C07304=1154.950,50.044,-50.253,-179.701,6.264,149.045
C07305=1154.955,49.796,-50.237,-179.703,6.263,149.046
C07306=1154.960,49.546,-50.222,-179.706,6.262,149.047
C07307=1154.965,49.296,-50.206,-179.708,6.261,149.047
C07308=1154.970,49.047,-50.190,-179.711,6.260,149.048
C07309=1154.975,48.798,-50.175,-179.714,6.259,149.048
C07310=1154.979,48.548,-50.159,-179.716,6.258,149.049
C07311=1154.985,48.298,-50.144,-179.719,6.257,149.049
C07312=1154.990,48.049,-50.128,-179.721,6.256,149.050
C07313=1154.996,47.800,-50.112,-179.724,6.255,149.050
C07314=1155.000,47.550,-50.097,-179.726,6.254,149.051
C07315=1155.005,47.300,-50.081,-179.730,6.252,149.051
C07316=1155.010,47.051,-50.066,-179.732,6.252,149.052
C07317=1155.015,46.802,-50.051,-179.734,6.251,149.052
C07318=1155.020,46.552,-50.035,-179.737,6.249,149.053
C07319=1155.025,46.302,-50.019,-179.739,6.249,149.053
C07320=1155.030,46.053,-50.004,-179.743,6.247,149.054
C07321=1155.035,45.804,-49.989,-179.745,6.246,149.055
C07322=1155.040,45.554,-49.973,-179.747,6.246,149.055
C07323=1155.045,45.305,-49.958,-179.750,6.244,149.056
C07324=1155.050,45.055,-49.942,-179.753,6.244,149.056
C07325=1155.055,44.806,-49.927,-179.756,6.242,149.057
C07326=1155.060,44.557,-49.912,-179.758,6.241,149.057
C07327=1155.065,44.307,-49.896,-179.760,6.241,149.058
C07328=1155.070,44.057,-49.880,-179.763,6.239,149.058
C07329=1155.075,43.808,-49.865,-179.766,6.239,149.059
C07330=1155.080,43.559,-49.849,-179.769,6.237,149.059
C07331=1155.086,43.309,-49.834,-179.771,6.237,149.060
C07332=1155.090,43.060,-49.819,-179.773,6.236,149.061
C07333=1155.095,42.810,-49.804,-179.777,6.234,149.061
C07334=1155.100,42.560,-49.789,-179.779,6.234,149.062
C07335=1155.105,42.311,-49.773,-179.781,6.232,149.062
C07336=1155.110,42.062,-49.758,-179.784,6.231,149.063
C07337=1155.116,41.813,-49.743,-179.786,6.231,149.063
C07338=1155.120,41.562,-49.727,-179.790,6.229,149.064
C07339=1155.125,41.313,-49.712,-179.792,6.228,149.064
C07340=1155.131,41.063,-49.697,-179.794,6.228,149.065
C07341=1155.135,40.814,-49.682,-179.797,6.226,149.066
C07342=1155.141,40.565,-49.666,-179.800,6.226,149.066
C07343=1155.145,40.316,-49.651,-179.802,6.224,149.067
C07344=1155.151,40.066,-49.636,-179.805,6.224,149.067
C07345=1155.156,39.817,-49.621,-179.807,6.223,149.068
C07346=1155.160,39.566,-49.605,-179.810,6.221,149.068
C07347=1155.165,39.317,-49.590,-179.813,6.221,149.069
C07348=1155.171,39.067,-49.575,-179.815,6.220,149.069
C07349=1155.175,38.818,-49.560,-179.818,6.219,149.070
C07350=1155.181,38.569,-49.545,-179.820,6.218,149.070
C07351=1155.185,38.320,-49.530,-179.823,6.217,149.071
C07352=1155.191,38.070,-49.515,-179.826,6.216,149.072
C07353=1155.196,37.821,-49.500,-179.828,6.215,149.072
C07354=1155.201,37.571,-49.484,-179.831,6.214,149.073
C07355=1155.206,37.322,-49.470,-179.834,6.213,149.073
C07356=1155.211,37.071,-49.454,-179.836,6.212,149.074
C07357=1155.216,36.822,-49.439,-179.839,6.211,149.074
C07358=1155.221,36.572,-49.424,-179.841,6.210,149.075
C07359=1155.226,36.323,-49.409,-179.843,6.209,149.075
C07360=1155.231,36.074,-49.395,-179.847,6.208,149.076
C07361=1155.236,35.824,-49.379,-179.849,6.207,149.077
C07362=1155.241,35.575,-49.364,-179.851,6.207,149.077
C07363=1155.247,35.325,-49.350,-179.854,6.205,149.078
C07364=1155.251,35.076,-49.335,-179.857,6.205,149.078
C07365=1155.256,34.826,-49.320,-179.859,6.204,149.079
C07366=1155.262,34.577,-49.305,-179.862,6.202,149.079
C07367=1155.266,34.328,-49.290,-179.864,6.202,149.080
C07368=1155.272,34.078,-49.275,-179.867,6.201,149.081
C07369=1155.277,33.829,-49.260,-179.870,6.200,149.081
C07370=1155.282,33.579,-49.246,-179.872,6.199,149.082
C07371=1155.287,33.330,-49.230,-179.875,6.198,149.082
C07372=1155.292,33.080,-49.216,-179.878,6.197,149.083
C07373=1155.297,32.831,-49.201,-179.880,6.196,149.083
C07374=1155.302,32.581,-49.186,-179.882,6.195,149.084
C07375=1155.307,32.332,-49.171,-179.885,6.194,149.084
C07376=1155.312,32.082,-49.157,-179.888,6.193,149.085
C07377=1155.317,31.833,-49.141,-179.890,6.193,149.086
C07378=1155.322,31.583,-49.127,-179.893,6.191,149.086
C07379=1155.327,31.334,-49.112,-179.896,6.191,149.087
C07380=1155.333,31.084,-49.097,-179.898,6.190,149.087
C07381=1155.337,30.834,-49.083,-179.900,6.189,149.088
C07382=1155.342,30.585,-49.068,-179.903,6.188,149.088
C07383=1155.347,30.335,-49.053,-179.906,6.187,149.089
C07384=1155.352,30.086,-49.038,-179.908,6.186,149.089
C07385=1155.357,29.836,-49.023,-179.911,6.185,149.090
C07386=1155.362,29.586,-49.009,-179.913,6.184,149.090
C07387=1155.367,29.337,-48.994,-179.916,6.184,149.091
C07388=1155.373,29.087,-48.979,-179.919,6.182,149.092
C07389=1155.377,28.838,-48.964,-179.921,6.182,149.092
C07390=1155.382,28.588,-48.950,-179.924,6.181,149.093
C07391=1155.387,28.339,-48.936,-179.926,6.180,149.093
C07392=1155.394,28.070,-48.920,-179.929,6.179,149.094
C07393=1155.399,27.802,-48.904,-179.932,6.178,149.095
C07394=1155.404,27.533,-48.888,-179.935,6.177,149.095
C07395=1155.410,27.264,-48.872,-179.937,6.176,149.096
C07396=1155.415,27.014,-48.858,-179.940,6.175,149.096
C07397=1155.420,26.764,-48.844,-179.942,6.174,149.097
C07398=1155.425,26.514,-48.829,-179.945,6.174,149.097
C07399=1155.429,26.265,-48.814,-179.947,6.173,149.098
C07400=1155.434,26.016,-48.800,-179.951,6.171,149.099
C07401=1155.440,25.766,-48.785,-179.953,6.171,149.099
C07402=1155.446,25.517,-48.771,-179.955,6.170,149.100
C07403=1155.450,25.268,-48.756,-179.958,6.169,149.100
C07404=1155.455,25.018,-48.742,-179.961,6.168,149.101
C07405=1155.460,24.768,-48.728,-179.963,6.167,149.101
C07406=1155.465,24.518,-48.713,-179.966,6.167,149.102
C07407=1155.470,24.269,-48.699,-179.968,6.165,149.102
C07408=1155.475,24.019,-48.684,-179.971,6.165,149.103
C07409=1155.481,23.770,-48.670,-179.973,6.164,149.104
C07410=1155.486,23.521,-48.655,-179.976,6.163,149.104
C07411=1155.491,23.271,-48.641,-179.979,6.162,149.105
C07412=1155.496,23.021,-48.627,-179.981,6.161,149.105
C07413=1155.501,22.771,-48.613,-179.983,6.160,149.106
C07414=1155.505,22.522,-48.598,-179.986,6.160,149.106
C07415=1155.511,22.273,-48.584,-179.989,6.158,149.107
C07416=1155.516,22.024,-48.569,-179.991,6.157,149.107
C07417=1155.521,21.774,-48.555,-179.994,6.157,149.108
C07418=1155.526,21.524,-48.541,-179.996,6.156,149.109
C07419=1155.531,21.275,-48.527,-179.999,6.155,149.109
C07420=1155.536,21.025,-48.512,179.999,6.154,149.110
C07421=1155.541,20.776,-48.498,179.996,6.154,149.110
C07422=1155.546,20.526,-48.484,179.994,6.153,149.111
C07423=1155.551,20.276,-48.470,179.991,6.152,149.112
C07424=1155.556,20.027,-48.455,179.989,6.151,149.112
C07425=1155.561,19.777,-48.441,179.986,6.150,149.113
C07426=1155.567,19.528,-48.427,179.984,6.149,149.113
C07427=1155.572,19.278,-48.413,179.981,6.148,149.114
C07428=1155.577,19.029,-48.399,179.978,6.147,149.114
C07429=1155.582,18.779,-48.384,179.976,6.147,149.115
C07430=1155.587,18.530,-48.371,179.974,6.146,149.115
C07431=1155.592,18.280,-48.356,179.970,6.145,149.116
C07432=1155.597,18.030,-48.342,179.968,6.144,149.117
C07433=1155.602,17.781,-48.328,179.965,6.143,149.117
C07434=1155.608,17.532,-48.314,179.963,6.143,149.118
C07435=1155.613,17.282,-48.300,179.961,6.142,149.118
C07436=1155.617,17.032,-48.285,179.958,6.141,149.119
C07437=1155.622,16.783,-48.271,179.955,6.140,149.120
C07438=1155.628,16.534,-48.257,179.953,6.139,149.120
C07439=1155.633,16.284,-48.243,179.950,6.139,149.121
C07440=1155.638,16.034,-48.229,179.948,6.137,149.121
C07441=1155.643,15.784,-48.214,179.945,6.137,149.122
C07442=1155.648,15.535,-48.200,179.943,6.136,149.122
C07443=1155.654,15.285,-48.187,179.940,6.135,149.123
C07444=1155.658,15.036,-48.173,179.938,6.135,149.123
C07445=1155.663,14.787,-48.159,179.935,6.133,149.124
C07446=1155.668,14.537,-48.145,179.933,6.133,149.125
C07447=1155.673,14.287,-48.131,179.930,6.132,149.125
C07448=1155.679,14.038,-48.117,179.928,6.131,149.126
C07449=1155.684,13.788,-48.103,179.925,6.131,149.126
C07450=1155.689,13.538,-48.089,179.922,6.129,149.127
C07451=1155.694,13.288,-48.075,179.920,6.129,149.128
C07452=1155.699,13.040,-48.061,179.918,6.128,149.128
C07453=1155.704,12.790,-48.047,179.915,6.127,149.129
C07454=1155.709,12.540,-48.033,179.913,6.127,149.129
C07455=1155.715,12.291,-48.020,179.910,6.125,149.130
C07456=1155.720,12.041,-48.005,179.907,6.125,149.130
C07457=1155.724,11.792,-47.992,179.905,6.124,149.131
C07458=1155.730,11.542,-47.978,179.903,6.123,149.131
C07459=1155.735,11.292,-47.964,179.900,6.123,149.132
C07460=1155.740,11.043,-47.950,179.897,6.121,149.133
C07461=1155.745,10.794,-47.936,179.894,6.121,149.133
C07462=1155.750,10.544,-47.923,179.892,6.120,149.134
C07463=1155.755,10.295,-47.909,179.890,6.119,149.134
C07464=1155.760,10.045,-47.895,179.887,6.119,149.135
C07465=1155.765,9.794,-47.881,179.885,6.118,149.136
C07466=1155.771,9.545,-47.867,179.882,6.117,149.136
C07467=1155.775,9.296,-47.854,179.879,6.116,149.137
C07468=1155.781,9.046,-47.840,179.877,6.115,149.137
C07469=1155.786,8.797,-47.826,179.875,6.115,149.138
C07470=1155.790,8.547,-47.812,179.872,6.114,149.138
C07471=1155.796,8.298,-47.799,179.870,6.114,149.139
C07472=1155.801,8.048,-47.785,179.867,6.112,149.139
C07473=1155.807,7.799,-47.771,179.864,6.111,149.140
C07474=1155.811,7.549,-47.758,179.862,6.111,149.141
C07475=1155.816,7.299,-47.744,179.859,6.110,149.141
C07476=1155.822,7.050,-47.731,179.857,6.109,149.142
C07477=1155.826,6.800,-47.717,179.855,6.109,149.142
C07478=1155.832,6.551,-47.703,179.852,6.107,149.143
C07479=1155.837,6.301,-47.689,179.849,6.107,149.144
C07480=1155.842,6.052,-47.676,179.847,6.106,149.144
C07481=1155.847,5.802,-47.663,179.844,6.106,149.145
C07482=1155.852,5.552,-47.648,179.842,6.105,149.145
C07483=1155.857,5.303,-47.636,179.840,6.104,149.146
C07484=1155.862,5.053,-47.621,179.837,6.103,149.146
C07485=1155.868,4.804,-47.608,179.834,6.102,149.147
C07486=1155.872,4.554,-47.595,179.832,6.101,149.147
C07487=1155.878,4.304,-47.581,179.829,6.101,149.148
C07488=1155.883,4.055,-47.567,179.827,6.100,149.149
C07489=1155.888,3.805,-47.554,179.825,6.100,149.149
C07490=1155.893,3.556,-47.540,179.822,6.099,149.150
C07491=1155.898,3.306,-47.528,179.820,6.098,149.150
C07492=1155.903,3.057,-47.513,179.816,6.097,149.151
C07493=1155.909,2.807,-47.500,179.814,6.096,149.152
C07494=1155.914,2.557,-47.487,179.812,6.096,149.152
C07495=1155.919,2.308,-47.473,179.809,6.095,149.153
C07496=1155.924,2.039,-47.459,179.807,6.095,149.153
C07497=1155.930,1.769,-47.445,179.804,6.093,149.154
C07498=1155.935,1.499,-47.430,179.801,6.093,149.155
C07499=1155.941,1.230,-47.416,179.799,6.092,149.155
C07500=1155.946,0.981,-47.402,179.797,6.091,149.156
C07501=1155.951,0.731,-47.389,179.794,6.091,149.156
C07502=1155.956,0.481,-47.376,179.791,6.089,149.157
C07503=1155.961,0.232,-47.362,179.788,6.089,149.158
C07504=1155.966,-0.018,-47.349,179.786,6.088,149.158
C07505=1155.972,-0.267,-47.335,179.784,6.088,149.159
C07506=1155.976,-0.517,-47.322,179.781,6.087,149.159
C07507=1155.982,-0.767,-47.309,179.779,6.086,149.160
C07508=1155.987,-1.016,-47.296,179.777,6.085,149.160
C07509=1155.992,-1.266,-47.282,179.774,6.085,149.161
C07510=1155.997,-1.515,-47.269,179.772,6.084,149.162
C07511=1156.002,-1.765,-47.256,179.769,6.083,149.162
C07512=1156.007,-2.014,-47.243,179.766,6.083,149.163
C07513=1156.012,-2.264,-47.229,179.764,6.082,149.163
C07514=1156.018,-2.514,-47.216,179.761,6.081,149.164
C07515=1156.023,-2.763,-47.203,179.759,6.080,149.165
C07516=1156.028,-3.013,-47.189,179.756,6.080,149.165
C07517=1156.034,-3.262,-47.176,179.754,6.079,149.166
C07518=1156.038,-3.512,-47.163,179.751,6.079,149.166
C07519=1156.044,-3.762,-47.150,179.749,6.078,149.167
C07520=1156.048,-4.011,-47.136,179.747,6.077,149.168
C07521=1156.053,-4.261,-47.124,179.744,6.076,149.168
C07522=1156.059,-4.510,-47.111,179.741,6.075,149.169
C07523=1156.064,-4.760,-47.098,179.739,6.075,149.169
C07524=1156.070,-5.010,-47.084,179.736,6.074,149.170
C07525=1156.075,-5.259,-47.072,179.734,6.073,149.170
C07526=1156.079,-5.509,-47.058,179.731,6.073,149.171
C07527=1156.085,-5.758,-47.045,179.729,6.072,149.171
C07528=1156.089,-6.008,-47.032,179.727,6.072,149.172
C07529=1156.095,-6.258,-47.019,179.724,6.071,149.173
C07530=1156.100,-6.507,-47.006,179.722,6.070,149.173
C07531=1156.105,-6.757,-46.993,179.720,6.070,149.174
C07532=1156.111,-7.007,-46.980,179.717,6.069,149.174
C07533=1156.115,-7.256,-46.967,179.714,6.068,149.175
C07534=1156.120,-7.506,-46.954,179.712,6.067,149.176
C07535=1156.126,-7.755,-46.941,179.709,6.066,149.176
C07536=1156.131,-8.005,-46.928,179.707,6.066,149.177
C07537=1156.135,-8.255,-46.915,179.705,6.065,149.177
C07538=1156.141,-8.504,-46.902,179.702,6.065,149.178
C07539=1156.146,-8.753,-46.889,179.700,6.064,149.178
C07540=1156.151,-9.003,-46.876,179.697,6.063,149.179
C07541=1156.157,-9.253,-46.863,179.695,6.063,149.180
C07542=1156.162,-9.502,-46.850,179.692,6.062,149.180
C07543=1156.166,-9.752,-46.838,179.690,6.061,149.181
C07544=1156.172,-10.002,-46.825,179.687,6.061,149.181
C07545=1156.177,-10.251,-46.812,179.685,6.060,149.182
C07546=1156.182,-10.501,-46.799,179.683,6.060,149.183
C07547=1156.187,-10.751,-46.786,179.680,6.059,149.183
C07548=1156.193,-11.000,-46.773,179.678,6.058,149.184
C07549=1156.198,-11.250,-46.760,179.675,6.057,149.184
C07550=1156.203,-11.500,-46.747,179.672,6.056,149.185
C07551=1156.208,-11.749,-46.735,179.670,6.056,149.186
C07552=1156.214,-11.999,-46.722,179.667,6.055,149.186
C07553=1156.218,-12.249,-46.709,179.665,6.055,149.187
C07554=1156.223,-12.498,-46.696,179.663,6.054,149.187
C07555=1156.228,-12.747,-46.683,179.660,6.053,149.188
C07556=1156.234,-12.997,-46.671,179.658,6.053,149.188
C07557=1156.239,-13.247,-46.657,179.655,6.052,149.189
C07558=1156.244,-13.497,-46.645,179.653,6.051,149.190
C07559=1156.249,-13.746,-46.633,179.650,6.051,149.190
C07560=1156.254,-13.996,-46.620,179.648,6.050,149.191
C07561=1156.259,-14.246,-46.607,179.645,6.050,149.191
C07562=1156.265,-14.495,-46.594,179.643,6.049,149.192
C07563=1156.270,-14.744,-46.581,179.641,6.048,149.193
C07564=1156.275,-14.994,-46.569,179.638,6.048,149.193
C07565=1156.281,-15.244,-46.557,179.636,6.047,149.194
C07566=1156.285,-15.494,-46.544,179.634,6.046,149.194
C07567=1156.290,-15.743,-46.531,179.631,6.046,149.195
C07568=1156.296,-15.993,-46.518,179.629,6.045,149.195
C07569=1156.301,-16.242,-46.506,179.626,6.045,149.196
C07570=1156.306,-16.492,-46.493,179.624,6.044,149.196
C07571=1156.311,-16.742,-46.481,179.621,6.043,149.197
C07572=1156.316,-16.991,-46.468,179.619,6.043,149.198
C07573=1156.321,-17.241,-46.456,179.616,6.042,149.198
C07574=1156.326,-17.490,-46.443,179.614,6.041,149.199
C07575=1156.331,-17.741,-46.431,179.612,6.041,149.199
C07576=1156.337,-17.990,-46.417,179.609,6.040,149.200
C07577=1156.342,-18.240,-46.405,179.607,6.040,149.201
C07578=1156.347,-18.489,-46.392,179.605,6.039,149.201
C07579=1156.353,-18.739,-46.380,179.602,6.038,149.202
C07580=1156.358,-18.988,-46.368,179.600,6.038,149.202
C07581=1156.362,-19.238,-46.355,179.597,6.037,149.203
C07582=1156.368,-19.488,-46.343,179.595,6.036,149.203
C07583=1156.373,-19.737,-46.330,179.592,6.036,149.204
C07584=1156.378,-19.987,-46.318,179.590,6.035,149.205
C07585=1156.384,-20.237,-46.306,179.587,6.035,149.205
C07586=1156.389,-20.486,-46.293,179.585,6.034,149.206
C07587=1156.394,-20.735,-46.281,179.583,6.034,149.206
C07588=1156.399,-20.986,-46.268,179.580,6.033,149.207
C07589=1156.404,-21.235,-46.256,179.578,6.032,149.208
C07590=1156.409,-21.485,-46.243,179.576,6.031,149.208
C07591=1156.414,-21.734,-46.231,179.573,6.031,149.209
C07592=1156.419,-21.984,-46.219,179.571,6.030,149.209
C07593=1156.425,-22.233,-46.206,179.568,6.030,149.210
C07594=1156.430,-22.483,-46.194,179.566,6.029,149.210
C07595=1156.435,-22.732,-46.182,179.563,6.029,149.211
C07596=1156.441,-22.982,-46.170,179.561,6.028,149.212
C07597=1156.446,-23.232,-46.157,179.558,6.027,149.212
C07598=1156.450,-23.482,-46.144,179.556,6.027,149.213
C07599=1156.456,-23.732,-46.132,179.553,6.026,149.213
C07600=1156.462,-24.002,-46.119,179.551,6.026,149.214
C07601=1156.467,-24.271,-46.105,179.549,6.025,149.215
C07602=1156.473,-24.542,-46.092,179.545,6.024,149.215
C07603=1156.478,-24.811,-46.079,179.543,6.023,149.216
C07604=1156.484,-25.061,-46.067,179.541,6.022,149.217
C07605=1156.489,-25.310,-46.055,179.538,6.022,149.217
C07606=1156.494,-25.560,-46.043,179.536,6.021,149.218
C07607=1156.499,-25.809,-46.030,179.533,6.021,149.218
C07608=1156.504,-26.060,-46.018,179.531,6.020,149.219
C07609=1156.509,-26.309,-46.005,179.528,6.020,149.220
C07610=1156.515,-26.559,-45.993,179.526,6.019,149.220
C07611=1156.520,-26.808,-45.981,179.524,6.019,149.221
C07612=1156.525,-27.058,-45.969,179.522,6.018,149.221
C07613=1156.530,-27.308,-45.956,179.519,6.018,149.222
C07614=1156.535,-27.557,-45.945,179.517,6.017,149.222
C07615=1156.540,-27.807,-45.933,179.514,6.017,149.223
C07616=1156.546,-28.056,-45.921,179.512,6.016,149.224
C07617=1156.551,-28.306,-45.909,179.509,6.015,149.224
C07618=1156.556,-28.556,-45.896,179.507,6.015,149.225
C07619=1156.562,-28.806,-45.884,179.505,6.014,149.225
C07620=1156.567,-29.056,-45.872,179.502,6.013,149.226
C07621=1156.571,-29.305,-45.860,179.500,6.013,149.227
C07622=1156.577,-29.555,-45.848,179.498,6.012,149.227
C07623=1156.582,-29.804,-45.836,179.495,6.012,149.228
C07624=1156.587,-30.054,-45.824,179.493,6.011,149.228
C07625=1156.593,-30.304,-45.812,179.490,6.011,149.229
C07626=1156.598,-30.553,-45.799,179.488,6.010,149.229
C07627=1156.603,-30.803,-45.788,179.485,6.009,149.230
C07628=1156.608,-31.053,-45.776,179.483,6.009,149.231
C07629=1156.613,-31.302,-45.764,179.480,6.008,149.231
C07630=1156.619,-31.552,-45.752,179.479,6.008,149.232
C07631=1156.623,-31.802,-45.740,179.476,6.008,149.232
C07632=1156.628,-32.051,-45.728,179.474,6.007,149.233
C07633=1156.634,-32.301,-45.716,179.471,6.006,149.234
C07634=1156.639,-32.551,-45.704,179.469,6.006,149.234
C07635=1156.645,-32.801,-45.692,179.466,6.005,149.235
C07636=1156.649,-33.050,-45.680,179.464,6.004,149.235
C07637=1156.655,-33.300,-45.668,179.462,6.004,149.236
C07638=1156.660,-33.550,-45.656,179.459,6.003,149.236
C07639=1156.666,-33.799,-45.645,179.457,6.003,149.237
C07640=1156.670,-34.048,-45.633,179.455,6.002,149.238
C07641=1156.676,-34.298,-45.621,179.452,6.002,149.238
C07642=1156.681,-34.548,-45.609,179.450,6.001,149.239
C07643=1156.687,-34.798,-45.597,179.447,6.000,149.239
C07644=1156.691,-35.047,-45.585,179.445,6.000,149.240
C07645=1156.696,-35.297,-45.573,179.443,6.000,149.241
C07646=1156.702,-35.546,-45.561,179.441,5.999,149.241
C07647=1156.707,-35.796,-45.550,179.438,5.999,149.242
C07648=1156.712,-36.046,-45.538,179.436,5.998,149.242
C07649=1156.717,-36.296,-45.526,179.433,5.998,149.243
C07650=1156.722,-36.545,-45.514,179.431,5.997,149.243
C07651=1156.728,-36.794,-45.503,179.428,5.996,149.244
C07652=1156.733,-37.044,-45.491,179.426,5.996,149.245
C07653=1156.738,-37.294,-45.480,179.423,5.995,149.245
C07654=1156.743,-37.544,-45.468,179.421,5.994,149.246
C07655=1156.749,-37.794,-45.456,179.419,5.995,149.246
C07656=1156.754,-38.043,-45.445,179.417,5.994,149.247
C07657=1156.759,-38.293,-45.433,179.414,5.993,149.248
C07658=1156.764,-38.543,-45.420,179.412,5.993,149.248
C07659=1156.769,-38.791,-45.409,179.409,5.992,149.249
C07660=1156.775,-39.041,-45.397,179.407,5.991,149.249
C07661=1156.780,-39.291,-45.385,179.405,5.991,149.250
C07662=1156.785,-39.541,-45.374,179.402,5.990,149.250
C07663=1156.790,-39.791,-45.362,179.400,5.990,149.251
C07664=1156.795,-40.040,-45.351,179.398,5.990,149.252
C07665=1156.801,-40.290,-45.339,179.395,5.989,149.252
C07666=1156.807,-40.540,-45.328,179.393,5.989,149.253
C07667=1156.811,-40.789,-45.316,179.391,5.988,149.254
C07668=1156.817,-41.039,-45.304,179.388,5.987,149.254
C07669=1156.821,-41.289,-45.293,179.386,5.987,149.255
C07670=1156.827,-41.539,-45.281,179.384,5.986,149.255
C07671=1156.833,-41.788,-45.270,179.381,5.986,149.256
C07672=1156.838,-42.038,-45.258,179.379,5.985,149.256
C07673=1156.843,-42.288,-45.247,179.377,5.985,149.257
C07674=1156.848,-42.537,-45.235,179.375,5.985,149.258
C07675=1156.853,-42.787,-45.223,179.372,5.984,149.258
C07676=1156.858,-43.037,-45.212,179.370,5.983,149.259
C07677=1156.864,-43.286,-45.201,179.367,5.983,149.259
C07678=1156.868,-43.536,-45.189,179.365,5.982,149.260
C07679=1156.874,-43.786,-45.177,179.362,5.982,149.261
C07680=1156.879,-44.035,-45.166,179.360,5.981,149.261
C07681=1156.885,-44.284,-45.155,179.358,5.981,149.262
C07682=1156.889,-44.534,-45.143,179.356,5.981,149.262
C07683=1156.895,-44.785,-45.132,179.354,5.980,149.263
C07684=1156.900,-45.034,-45.121,179.351,5.979,149.263
C07685=1156.905,-45.284,-45.109,179.349,5.979,149.264
C07686=1156.910,-45.533,-45.098,179.346,5.978,149.265
C07687=1156.916,-45.783,-45.086,179.344,5.977,149.265
C07688=1156.921,-46.033,-45.075,179.342,5.978,149.266
C07689=1156.926,-46.283,-45.063,179.340,5.977,149.266
C07690=1156.931,-46.532,-45.052,179.337,5.977,149.267
C07691=1156.937,-46.782,-45.041,179.335,5.976,149.267
C07692=1156.942,-47.032,-45.030,179.332,5.975,149.268
C07693=1156.947,-47.282,-45.018,179.330,5.975,149.269
C07694=1156.952,-47.531,-45.007,179.327,5.974,149.269
C07695=1156.958,-47.780,-44.995,179.326,5.974,149.270
C07696=1156.963,-48.031,-44.984,179.323,5.974,149.270
C07697=1156.968,-48.280,-44.973,179.321,5.973,149.271
C07698=1156.974,-48.530,-44.962,179.318,5.973,149.272
C07699=1156.978,-48.779,-44.950,179.316,5.972,149.272
C07700=1156.984,-49.029,-44.938,179.313,5.971,149.273
C07701=1156.989,-49.279,-44.928,179.312,5.971,149.273
C07702=1156.994,-49.528,-44.917,179.309,5.971,149.274
C07703=1156.999,-49.778,-44.905,179.307,5.970,149.275
C07704=1157.006,-50.049,-44.893,179.304,5.970,149.275
C07705=1157.011,-50.320,-44.881,179.302,5.969,149.276
C07706=1157.016,-50.590,-44.869,179.299,5.969,149.276
C07707=1157.022,-50.860,-44.857,179.297,5.968,149.277
C07708=1157.028,-51.110,-44.845,179.294,5.967,149.278
C07709=1157.032,-51.360,-44.834,179.292,5.967,149.278
C07710=1157.038,-51.609,-44.823,179.290,5.966,149.279
C07711=1157.044,-51.860,-44.812,179.287,5.967,149.279
C07712=1157.048,-52.109,-44.801,179.285,5.966,149.280
C07713=1157.054,-52.358,-44.790,179.283,5.965,149.281
C07714=1157.059,-52.609,-44.779,179.280,5.965,149.281
C07715=1157.064,-52.858,-44.767,179.278,5.964,149.282
C07716=1157.069,-53.107,-44.756,179.276,5.963,149.282
C07717=1157.075,-53.358,-44.745,179.274,5.963,149.283
C07718=1157.080,-53.607,-44.734,179.271,5.963,149.283
C07719=1157.085,-53.856,-44.723,179.269,5.962,149.284
C07720=1157.091,-54.107,-44.712,179.266,5.962,149.285
C07721=1157.095,-54.356,-44.701,179.264,5.961,149.285
C07722=1157.101,-54.605,-44.690,179.262,5.961,149.286
C07723=1157.106,-54.856,-44.679,179.260,5.961,149.286
C07724=1157.112,-55.105,-44.668,179.257,5.960,149.287
C07725=1157.117,-55.355,-44.657,179.255,5.959,149.288
C07726=1157.121,-55.605,-44.646,179.252,5.959,149.288
C07727=1157.127,-55.854,-44.635,179.251,5.959,149.289
C07728=1157.132,-56.104,-44.624,179.249,5.958,149.289
C07729=1157.137,-56.354,-44.612,179.246,5.958,149.290
C07730=1157.143,-56.603,-44.602,179.244,5.957,149.290
C07731=1157.147,-56.853,-44.591,179.241,5.957,149.291
C07732=1157.154,-57.103,-44.580,179.240,5.957,149.292
C07733=1157.158,-57.352,-44.569,179.237,5.956,149.292
C07734=1157.163,-57.603,-44.558,179.235,5.955,149.293
C07735=1157.169,-57.852,-44.547,179.232,5.955,149.293
C07736=1157.174,-58.102,-44.537,179.230,5.954,149.294
C07737=1157.180,-58.351,-44.525,179.228,5.955,149.295
C07738=1157.185,-58.601,-44.515,179.226,5.954,149.295
C07739=1157.189,-58.851,-44.503,179.223,5.953,149.296
C07740=1157.195,-59.101,-44.493,179.221,5.953,149.296
C07741=1157.200,-59.350,-44.482,179.219,5.952,149.297
C07742=1157.206,-59.600,-44.471,179.217,5.952,149.297
C07743=1157.211,-59.850,-44.460,179.214,5.952,149.298
C07744=1157.216,-60.099,-44.449,179.212,5.951,149.299
C07745=1157.221,-60.349,-44.438,179.209,5.950,149.299
C07746=1157.227,-60.598,-44.428,179.207,5.950,149.300
C07747=1157.232,-60.849,-44.417,179.205,5.950,149.300
C07748=1157.236,-61.098,-44.406,179.203,5.950,149.301
C07749=1157.243,-61.348,-44.395,179.200,5.949,149.301
C07750=1157.247,-61.598,-44.384,179.198,5.948,149.302
C07751=1157.253,-61.847,-44.374,179.196,5.948,149.303
C07752=1157.258,-62.098,-44.363,179.194,5.948,149.303
C07753=1157.263,-62.346,-44.352,179.191,5.947,149.304
C07754=1157.268,-62.597,-44.342,179.189,5.946,149.304
C07755=1157.274,-62.846,-44.331,179.186,5.946,149.305
C07756=1157.279,-63.096,-44.320,179.185,5.946,149.306
C07757=1157.285,-63.346,-44.309,179.182,5.946,149.306
C07758=1157.290,-63.595,-44.298,179.180,5.945,149.307
C07759=1157.295,-63.845,-44.288,179.178,5.944,149.307
C07760=1157.300,-64.095,-44.277,179.176,5.944,149.308
C07761=1157.305,-64.344,-44.266,179.173,5.944,149.308
C07762=1157.310,-64.594,-44.256,179.171,5.943,149.309
C07763=1157.316,-64.844,-44.246,179.169,5.943,149.310
C07764=1157.321,-65.094,-44.235,179.167,5.943,149.310
C07765=1157.326,-65.343,-44.224,179.164,5.942,149.311
C07766=1157.331,-65.593,-44.214,179.162,5.941,149.311
C07767=1157.337,-65.843,-44.203,179.159,5.941,149.312
C07768=1157.342,-66.092,-44.192,179.158,5.941,149.312
C07769=1157.347,-66.342,-44.182,179.155,5.941,149.313
C07770=1157.352,-66.592,-44.171,179.153,5.940,149.314
C07771=1157.358,-66.842,-44.161,179.150,5.939,149.314
C07772=1157.363,-67.091,-44.150,179.148,5.939,149.315
C07773=1157.368,-67.341,-44.140,179.147,5.939,149.315
C07774=1157.374,-67.590,-44.129,179.144,5.938,149.316
C07775=1157.379,-67.841,-44.118,179.142,5.937,149.316
C07776=1157.385,-68.090,-44.107,179.140,5.938,149.317
C07777=1157.390,-68.340,-44.097,179.137,5.937,149.318
C07778=1157.395,-68.590,-44.086,179.135,5.937,149.318
C07779=1157.400,-68.840,-44.076,179.133,5.936,149.319
C07780=1157.405,-69.089,-44.066,179.131,5.936,149.319
C07781=1157.411,-69.339,-44.056,179.128,5.936,149.320
C07782=1157.415,-69.588,-44.045,179.126,5.935,149.320
C07783=1157.421,-69.838,-44.035,179.123,5.934,149.321
C07784=1157.426,-70.088,-44.024,179.122,5.934,149.322
C07785=1157.432,-70.338,-44.014,179.119,5.934,149.322
C07786=1157.437,-70.587,-44.004,179.117,5.933,149.323
C07787=1157.442,-70.837,-43.993,179.115,5.932,149.323
C07788=1157.448,-71.086,-43.982,179.113,5.933,149.324
C07789=1157.453,-71.337,-43.972,179.111,5.932,149.325
C07790=1157.458,-71.586,-43.961,179.108,5.932,149.325
C07791=1157.464,-71.836,-43.951,179.106,5.931,149.326
C07792=1157.469,-72.086,-43.941,179.104,5.931,149.326
C07793=1157.474,-72.336,-43.930,179.101,5.930,149.327
C07794=1157.479,-72.586,-43.920,179.099,5.930,149.327
C07795=1157.485,-72.835,-43.910,179.097,5.930,149.328
C07796=1157.491,-73.085,-43.899,179.095,5.929,149.329
C07797=1157.496,-73.335,-43.889,179.092,5.929,149.329
C07798=1157.500,-73.584,-43.879,179.090,5.928,149.330
C07799=1157.506,-73.834,-43.869,179.089,5.928,149.330
C07800=1157.511,-74.084,-43.858,179.086,5.928,149.331
C07801=1157.516,-74.333,-43.847,179.084,5.927,149.331
C07802=1157.522,-74.583,-43.837,179.082,5.927,149.332
C07803=1157.527,-74.833,-43.827,179.079,5.927,149.333
C07804=1157.532,-75.082,-43.816,179.077,5.926,149.333
C07805=1157.538,-75.332,-43.806,179.075,5.925,149.334
C07806=1157.542,-75.582,-43.796,179.073,5.925,149.334
C07807=1157.548,-75.831,-43.786,179.070,5.925,149.335
C07808=1157.554,-76.103,-43.775,179.068,5.924,149.335
C07809=1157.560,-76.374,-43.765,179.065,5.924,149.336
C07810=1157.566,-76.646,-43.753,179.063,5.923,149.337
C07811=1157.571,-76.917,-43.742,179.061,5.924,149.337
C07812=1157.577,-77.167,-43.732,179.059,5.923,149.338
C07813=1157.582,-77.416,-43.722,179.056,5.922,149.339
C07814=1157.587,-77.666,-43.711,179.054,5.922,149.339
C07815=1157.593,-77.916,-43.701,179.052,5.922,149.340
C07816=1157.598,-78.165,-43.691,179.050,5.921,149.340
C07817=1157.603,-78.415,-43.681,179.048,5.920,149.341
C07818=1157.608,-78.665,-43.671,179.046,5.921,149.341
C07819=1157.614,-78.915,-43.660,179.043,5.920,149.342
C07820=1157.620,-79.164,-43.650,179.041,5.920,149.343
C07821=1157.624,-79.414,-43.640,179.039,5.920,149.343
C07822=1157.630,-79.664,-43.631,179.037,5.919,149.344
C07823=1157.635,-79.914,-43.620,179.034,5.919,149.344
C07824=1157.640,-80.164,-43.610,179.033,5.919,149.345
C07825=1157.645,-80.413,-43.600,179.030,5.918,149.346
C07826=1157.651,-80.663,-43.590,179.028,5.917,149.346
C07827=1157.656,-80.912,-43.580,179.026,5.917,149.346
C07828=1157.661,-81.163,-43.569,179.024,5.917,149.347
C07829=1157.666,-81.412,-43.560,179.021,5.916,149.348
C07830=1157.672,-81.662,-43.550,179.019,5.916,149.348
C07831=1157.678,-81.911,-43.540,179.017,5.916,149.349
C07832=1157.683,-82.162,-43.529,179.015,5.915,149.349
C07833=1157.688,-82.411,-43.520,179.012,5.915,149.350
C07834=1157.693,-82.660,-43.510,179.011,5.915,149.351
C07835=1157.699,-82.911,-43.500,179.008,5.914,149.351
C07836=1157.703,-83.161,-43.490,179.006,5.914,149.352
C07837=1157.709,-83.410,-43.480,179.004,5.914,149.352
C07838=1157.715,-83.660,-43.470,179.001,5.913,149.353
C07839=1157.720,-83.910,-43.461,178.999,5.913,149.353
C07840=1157.725,-84.160,-43.450,178.998,5.913,149.354
C07841=1157.730,-84.409,-43.440,178.995,5.912,149.355
C07842=1157.735,-84.659,-43.430,178.993,5.911,149.355
C07843=1157.741,-84.909,-43.421,178.991,5.911,149.356
C07844=1157.747,-85.158,-43.411,178.989,5.911,149.356
C07845=1157.751,-85.408,-43.401,178.986,5.910,149.357
C07846=1157.756,-85.658,-43.391,178.984,5.911,149.357
C07847=1157.762,-85.908,-43.381,178.982,5.910,149.358
C07848=1157.767,-86.157,-43.371,178.980,5.909,149.358
C07849=1157.773,-86.407,-43.361,178.978,5.910,149.359
C07850=1157.778,-86.657,-43.351,178.976,5.909,149.360
C07851=1157.783,-86.907,-43.342,178.973,5.908,149.360
C07852=1157.789,-87.156,-43.332,178.971,5.908,149.361
C07853=1157.793,-87.406,-43.322,178.969,5.908,149.361
C07854=1157.799,-87.656,-43.312,178.966,5.907,149.362
C07855=1157.804,-87.906,-43.302,178.965,5.907,149.362
C07856=1157.809,-88.155,-43.292,178.963,5.907,149.363
C07857=1157.815,-88.405,-43.283,178.960,5.906,149.364
C07858=1157.820,-88.655,-43.273,178.958,5.906,149.364
C07859=1157.826,-88.905,-43.264,178.956,5.905,149.365
C07860=1157.832,-89.154,-43.253,178.954,5.905,149.365
C07861=1157.836,-89.404,-43.244,178.952,5.905,149.366
C07862=1157.842,-89.654,-43.234,178.950,5.904,149.366
C07863=1157.847,-89.904,-43.224,178.948,5.905,149.367
C07864=1157.852,-90.154,-43.215,178.946,5.904,149.368
C07865=1157.857,-90.403,-43.205,178.943,5.903,149.368
C07866=1157.863,-90.653,-43.195,178.941,5.904,149.369
C07867=1157.868,-90.902,-43.186,178.939,5.903,149.369
C07868=1157.874,-91.152,-43.176,178.937,5.902,149.370
C07869=1157.879,-91.403,-43.166,178.935,5.902,149.370
C07870=1157.884,-91.652,-43.156,178.933,5.902,149.371
C07871=1157.890,-91.902,-43.147,178.930,5.901,149.372
C07872=1157.895,-92.151,-43.137,178.928,5.901,149.372
C07873=1157.900,-92.401,-43.127,178.926,5.901,149.373
C07874=1157.905,-92.651,-43.118,178.923,5.900,149.373
C07875=1157.911,-92.900,-43.108,178.922,5.900,149.374
C07876=1157.916,-93.150,-43.099,178.920,5.899,149.374
C07877=1157.922,-93.400,-43.089,178.918,5.900,149.375
C07878=1157.926,-93.650,-43.080,178.915,5.899,149.375
C07879=1157.932,-93.900,-43.069,178.913,5.898,149.376
C07880=1157.937,-94.150,-43.061,178.911,5.899,149.377
C07881=1157.943,-94.399,-43.050,178.909,5.898,149.377
C07882=1157.948,-94.649,-43.041,178.907,5.897,149.378
C07883=1157.953,-94.899,-43.031,178.905,5.898,149.378
C07884=1157.959,-95.148,-43.022,178.902,5.897,149.379
C07885=1157.964,-95.398,-43.013,178.901,5.897,149.379
C07886=1157.969,-95.648,-43.003,178.898,5.896,149.380
C07887=1157.975,-95.898,-42.994,178.896,5.896,149.380
C07888=1157.980,-96.147,-42.984,178.894,5.896,149.381
C07889=1157.985,-96.397,-42.975,178.892,5.895,149.382
C07890=1157.991,-96.647,-42.965,178.890,5.895,149.382
C07891=1157.996,-96.897,-42.956,178.888,5.895,149.383
C07892=1158.002,-97.147,-42.947,178.885,5.894,149.383
C07893=1158.007,-97.396,-42.937,178.884,5.894,149.384
C07894=1158.011,-97.646,-42.928,178.881,5.893,149.384
C07895=1158.017,-97.896,-42.918,178.879,5.893,149.385
C07896=1158.022,-98.146,-42.909,178.877,5.893,149.386
C07897=1158.028,-98.396,-42.899,178.875,5.892,149.386
C07898=1158.033,-98.645,-42.890,178.873,5.892,149.386
C07899=1158.038,-98.895,-42.881,178.871,5.892,149.387
C07900=1158.044,-99.145,-42.871,178.869,5.891,149.388
C07901=1158.049,-99.395,-42.862,178.867,5.891,149.388
C07902=1158.055,-99.645,-42.852,178.864,5.891,149.389
C07903=1158.060,-99.895,-42.843,178.863,5.891,149.389
C07904=1158.065,-100.144,-42.834,178.860,5.890,149.390
C07905=1158.071,-100.394,-42.824,178.858,5.890,149.391
C07906=1158.076,-100.644,-42.815,178.856,5.890,149.391
C07907=1158.081,-100.893,-42.806,178.854,5.889,149.392
C07908=1158.087,-101.143,-42.796,178.852,5.889,149.392
C07909=1158.092,-101.393,-42.787,178.850,5.889,149.393
C07910=1158.097,-101.642,-42.777,178.848,5.888,149.393
C07911=1158.103,-101.892,-42.768,178.845,5.888,149.394
C07912=1158.108,-102.164,-42.758,178.843,5.888,149.394
C07913=1158.114,-102.436,-42.749,178.841,5.887,149.395
C07914=1158.120,-102.708,-42.738,178.839,5.887,149.396
C07915=1158.125,-102.980,-42.728,178.836,5.887,149.396
C07916=1158.131,-103.230,-42.719,178.834,5.886,149.397
C07917=1158.136,-103.479,-42.709,178.833,5.886,149.397
C07918=1158.141,-103.729,-42.700,178.830,5.885,149.398
C07919=1158.147,-103.979,-42.691,178.828,5.886,149.398
C07920=1158.152,-104.229,-42.682,178.826,5.885,149.399
C07921=1158.158,-104.479,-42.673,178.824,5.884,149.399
C07922=1158.162,-104.728,-42.663,178.822,5.885,149.400
C07923=1158.168,-104.979,-42.654,178.820,5.884,149.401
C07924=1158.174,-105.228,-42.645,178.818,5.884,149.401
C07925=1158.179,-105.478,-42.636,178.816,5.883,149.402
C07926=1158.184,-105.727,-42.627,178.813,5.883,149.402
C07927=1158.190,-105.977,-42.617,178.812,5.883,149.403
C07928=1158.195,-106.227,-42.608,178.809,5.882,149.403
C07929=1158.200,-106.477,-42.599,178.807,5.883,149.404
C07930=1158.206,-106.726,-42.591,178.805,5.882,149.405
C07931=1158.211,-106.977,-42.581,178.803,5.882,149.405
C07932=1158.217,-107.227,-42.572,178.801,5.881,149.405
C07933=1158.222,-107.476,-42.563,178.799,5.881,149.406
C07934=1158.227,-107.726,-42.554,178.797,5.881,149.407
C07935=1158.233,-107.976,-42.544,178.795,5.880,149.407
C07936=1158.238,-108.226,-42.535,178.793,5.880,149.408
C07937=1158.243,-108.475,-42.526,178.791,5.880,149.408
C07938=1158.249,-108.725,-42.518,178.789,5.880,149.409
C07939=1158.254,-108.974,-42.509,178.787,5.879,149.409
C07940=1158.260,-109.225,-42.499,178.785,5.879,149.410
C07941=1158.265,-109.474,-42.491,178.782,5.879,149.411
C07942=1158.270,-109.724,-42.482,178.780,5.878,149.411
C07943=1158.275,-109.974,-42.473,178.779,5.878,149.412
C07944=1158.280,-110.223,-42.463,178.776,5.877,149.412
C07945=1158.285,-110.473,-42.454,178.774,5.877,149.413
C07946=1158.291,-110.723,-42.445,178.772,5.877,149.413
C07947=1158.297,-110.973,-42.436,178.770,5.877,149.414
C07948=1158.302,-111.222,-42.427,178.768,5.876,149.414
C07949=1158.307,-111.472,-42.418,178.766,5.876,149.415
C07950=1158.312,-111.722,-42.410,178.764,5.876,149.415
C07951=1158.318,-111.972,-42.401,178.761,5.875,149.416
C07952=1158.323,-112.222,-42.391,178.760,5.875,149.417
C07953=1158.329,-112.472,-42.382,178.758,5.875,149.417
C07954=1158.334,-112.721,-42.374,178.756,5.875,149.418
C07955=1158.340,-112.971,-42.365,178.753,5.874,149.418
C07956=1158.345,-113.221,-42.356,178.752,5.874,149.419
C07957=1158.350,-113.471,-42.347,178.750,5.874,149.419
C07958=1158.355,-113.721,-42.338,178.748,5.874,149.420
C07959=1158.360,-113.970,-42.329,178.745,5.873,149.420
C07960=1158.366,-114.220,-42.321,178.743,5.872,149.421
C07961=1158.372,-114.470,-42.311,178.742,5.872,149.421
C07962=1158.377,-114.720,-42.302,178.739,5.872,149.422
C07963=1158.382,-114.969,-42.293,178.737,5.872,149.423
C07964=1158.388,-115.220,-42.285,178.735,5.871,149.423
C07965=1158.393,-115.469,-42.277,178.733,5.871,149.424
C07966=1158.399,-115.719,-42.268,178.731,5.871,149.424
C07967=1158.404,-115.969,-42.259,178.730,5.871,149.425
C07968=1158.409,-116.219,-42.250,178.727,5.870,149.425
C07969=1158.414,-116.468,-42.241,178.725,5.870,149.426
C07970=1158.420,-116.718,-42.233,178.723,5.870,149.426
C07971=1158.425,-116.967,-42.224,178.722,5.870,149.427
C07972=1158.430,-117.217,-42.215,178.719,5.869,149.427
C07973=1158.435,-117.467,-42.206,178.717,5.868,149.428
C07974=1158.441,-117.718,-42.198,178.715,5.869,149.428
C07975=1158.447,-117.967,-42.189,178.713,5.868,149.429
C07976=1158.453,-118.217,-42.180,178.711,5.868,149.430
C07977=1158.458,-118.467,-42.171,178.709,5.867,149.430
C07978=1158.463,-118.717,-42.162,178.707,5.867,149.431
C07979=1158.469,-118.966,-42.153,178.705,5.867,149.431
C07980=1158.474,-119.216,-42.144,178.703,5.867,149.432
C07981=1158.479,-119.466,-42.136,178.701,5.866,149.432
C07982=1158.484,-119.716,-42.127,178.699,5.866,149.433
C07983=1158.490,-119.966,-42.118,178.697,5.866,149.433
C07984=1158.495,-120.215,-42.110,178.695,5.866,149.434
C07985=1158.501,-120.465,-42.101,178.693,5.865,149.434
C07986=1158.506,-120.715,-42.093,178.691,5.865,149.435
C07987=1158.510,-120.965,-42.085,178.689,5.865,149.435
C07988=1158.516,-121.214,-42.076,178.687,5.865,149.436
C07989=1158.521,-121.464,-42.067,178.685,5.864,149.436
C07990=1158.527,-121.714,-42.058,178.683,5.864,149.437
C07991=1158.533,-121.963,-42.050,178.681,5.864,149.438
C07992=1158.538,-122.213,-42.041,178.679,5.864,149.438
C07993=1158.543,-122.463,-42.033,178.677,5.863,149.439
C07994=1158.548,-122.713,-42.024,178.675,5.863,149.439
C07995=1158.554,-122.963,-42.016,178.673,5.863,149.440
C07996=1158.559,-123.213,-42.007,178.671,5.863,149.440
C07997=1158.565,-123.462,-41.998,178.669,5.862,149.441
C07998=1158.570,-123.712,-41.989,178.667,5.862,149.441
C07999=1158.576,-123.962,-41.981,178.665,5.861,149.442
C08000=1158.581,-124.212,-41.972,178.663,5.862,149.442
C08001=1158.586,-124.462,-41.964,178.661,5.861,149.443
C08002=1158.592,-124.712,-41.956,178.659,5.860,149.443
C08003=1158.597,-124.961,-41.947,178.657,5.860,149.444
C08004=1158.602,-125.211,-41.939,178.655,5.859,149.444
C08005=1158.608,-125.461,-41.931,178.653,5.859,149.445
C08006=1158.613,-125.711,-41.922,178.650,5.859,149.446
C08007=1158.618,-125.960,-41.913,178.649,5.859,149.446
C08008=1158.624,-126.210,-41.905,178.647,5.858,149.447
C08009=1158.629,-126.460,-41.896,178.645,5.858,149.447
C08010=1158.635,-126.710,-41.887,178.643,5.858,149.448
C08011=1158.641,-126.960,-41.880,178.641,5.858,149.448
C08012=1158.645,-127.209,-41.871,178.639,5.858,149.449
C08013=1158.650,-127.459,-41.862,178.637,5.857,149.449
C08014=1158.656,-127.709,-41.854,178.635,5.857,149.450
C08015=1158.662,-127.959,-41.846,178.633,5.857,149.450
C08016=1158.240,-127.970,-41.888,178.629,5.860,149.452
C08017=1158.235,-127.720,-41.896,178.632,5.861,149.452
C08018=1158.230,-127.471,-41.904,178.633,5.861,149.451
C08019=1158.224,-127.220,-41.912,178.635,5.861,149.451
C08020=1158.219,-126.971,-41.921,178.637,5.861,149.450
C08021=1158.213,-126.721,-41.930,178.640,5.862,149.449
C08022=1158.208,-126.471,-41.938,178.641,5.862,149.449
C08023=1158.203,-126.221,-41.947,178.643,5.862,149.448
C08024=1158.197,-125.972,-41.955,178.645,5.862,149.448
C08025=1158.191,-125.721,-41.964,178.647,5.863,149.447
C08026=1158.187,-125.472,-41.972,178.649,5.863,149.447
C08027=1158.181,-125.223,-41.980,178.651,5.863,149.446
C08028=1158.176,-124.972,-41.989,178.653,5.863,149.446
C08029=1158.171,-124.722,-41.997,178.655,5.864,149.445
C08030=1158.165,-124.473,-42.006,178.657,5.864,149.445
C08031=1158.159,-124.223,-42.014,178.660,5.864,149.444
C08032=1158.154,-123.973,-42.023,178.661,5.864,149.444
C08033=1158.149,-123.723,-42.032,178.663,5.865,149.443
C08034=1158.143,-123.474,-42.041,178.665,5.865,149.443
C08035=1158.138,-123.223,-42.049,178.667,5.866,149.442
C08036=1158.133,-122.974,-42.058,178.669,5.865,149.441
C08037=1158.127,-122.724,-42.067,178.671,5.866,149.441
C08038=1158.122,-122.474,-42.074,178.673,5.866,149.440
C08039=1158.117,-122.224,-42.083,178.675,5.867,149.440
C08040=1158.112,-121.975,-42.092,178.677,5.867,149.439
C08041=1158.106,-121.725,-42.100,178.679,5.867,149.439
C08042=1158.101,-121.476,-42.109,178.681,5.867,149.438
C08043=1158.095,-121.225,-42.117,178.683,5.868,149.438
C08044=1158.090,-120.975,-42.126,178.685,5.869,149.437
C08045=1158.084,-120.726,-42.135,178.687,5.869,149.437
C08046=1158.079,-120.476,-42.143,178.690,5.869,149.436
C08047=1158.074,-120.226,-42.152,178.691,5.869,149.436
C08048=1158.069,-119.976,-42.161,178.694,5.870,149.435
C08049=1158.063,-119.727,-42.169,178.695,5.870,149.435
C08050=1158.058,-119.477,-42.178,178.697,5.870,149.434
C08051=1158.053,-119.227,-42.187,178.699,5.870,149.433
C08052=1158.047,-118.977,-42.196,178.702,5.871,149.433
C08053=1158.041,-118.727,-42.204,178.703,5.871,149.432
C08054=1158.036,-118.478,-42.212,178.705,5.871,149.432
C08055=1158.031,-118.228,-42.221,178.707,5.871,149.431
C08056=1158.026,-117.978,-42.230,178.710,5.872,149.431
C08057=1158.021,-117.728,-42.239,178.711,5.872,149.430
C08058=1158.015,-117.479,-42.248,178.713,5.873,149.430
C08059=1158.010,-117.229,-42.257,178.715,5.872,149.429
C08060=1158.004,-116.979,-42.265,178.718,5.873,149.429
C08061=1157.999,-116.729,-42.274,178.719,5.873,149.428
C08062=1157.993,-116.480,-42.282,178.722,5.874,149.428
C08063=1157.988,-116.230,-42.291,178.724,5.874,149.427
C08064=1157.983,-115.980,-42.300,178.725,5.874,149.427
C08065=1157.977,-115.730,-42.310,178.728,5.875,149.426
C08066=1157.972,-115.480,-42.318,178.730,5.875,149.425
C08067=1157.966,-115.231,-42.327,178.732,5.875,149.425
C08068=1157.961,-114.981,-42.336,178.733,5.875,149.424
C08069=1157.956,-114.731,-42.345,178.736,5.876,149.424
C08070=1157.951,-114.481,-42.354,178.738,5.876,149.423
C08071=1157.946,-114.231,-42.363,178.740,5.876,149.423
C08072=1157.940,-113.981,-42.371,178.741,5.876,149.422
C08073=1157.934,-113.732,-42.379,178.744,5.877,149.422
C08074=1157.929,-113.482,-42.388,178.746,5.877,149.421
C08075=1157.923,-113.232,-42.398,178.748,5.878,149.421
C08076=1157.918,-112.982,-42.407,178.750,5.878,149.420
C08077=1157.913,-112.732,-42.415,178.752,5.878,149.419
C08078=1157.908,-112.482,-42.424,178.754,5.879,149.419
C08079=1157.902,-112.233,-42.433,178.756,5.879,149.418
C08080=1157.897,-111.983,-42.442,178.758,5.879,149.418
C08081=1157.892,-111.733,-42.451,178.760,5.879,149.417
C08082=1157.886,-111.483,-42.460,178.762,5.880,149.417
C08083=1157.881,-111.233,-42.469,178.764,5.880,149.416
C08084=1157.875,-110.983,-42.478,178.766,5.880,149.416
C08085=1157.870,-110.734,-42.486,178.769,5.881,149.415
C08086=1157.865,-110.485,-42.496,178.771,5.881,149.415
C08087=1157.860,-110.235,-42.505,178.773,5.881,149.414
C08088=1157.854,-109.985,-42.514,178.774,5.881,149.414
C08089=1157.848,-109.735,-42.523,178.777,5.882,149.413
C08090=1157.843,-109.485,-42.532,178.779,5.882,149.412
C08091=1157.838,-109.235,-42.541,178.781,5.883,149.412
C08092=1157.833,-108.986,-42.550,178.782,5.883,149.411
C08093=1157.828,-108.736,-42.559,178.785,5.883,149.411
C08094=1157.821,-108.486,-42.568,178.787,5.884,149.410
C08095=1157.816,-108.236,-42.577,178.789,5.884,149.410
C08096=1157.811,-107.987,-42.586,178.792,5.884,149.409
C08097=1157.806,-107.737,-42.595,178.793,5.884,149.409
C08098=1157.801,-107.488,-42.604,178.795,5.885,149.408
C08099=1157.795,-107.237,-42.614,178.797,5.885,149.408
C08100=1157.790,-106.988,-42.623,178.800,5.885,149.407
C08101=1157.785,-106.738,-42.632,178.802,5.886,149.406
C08102=1157.780,-106.488,-42.641,178.803,5.886,149.406
C08103=1157.774,-106.238,-42.650,178.806,5.887,149.405
C08104=1157.768,-105.988,-42.659,178.808,5.886,149.405
C08105=1157.764,-105.739,-42.669,178.810,5.887,149.404
C08106=1157.758,-105.489,-42.677,178.811,5.887,149.404
C08107=1157.752,-105.239,-42.687,178.814,5.887,149.403
C08108=1157.747,-104.989,-42.696,178.816,5.888,149.402
C08109=1157.742,-104.740,-42.704,178.818,5.888,149.402
C08110=1157.737,-104.490,-42.714,178.820,5.889,149.402
C08111=1157.731,-104.240,-42.724,178.822,5.888,149.401
C08112=1157.726,-103.990,-42.732,178.824,5.889,149.400
C08113=1157.721,-103.740,-42.741,178.827,5.890,149.400
C08114=1157.716,-103.491,-42.751,178.829,5.889,149.399
C08115=1157.710,-103.241,-42.760,178.831,5.890,149.399
C08116=1157.705,-102.991,-42.769,178.832,5.890,149.398
C08117=1157.699,-102.719,-42.780,178.835,5.891,149.397
C08118=1157.693,-102.447,-42.789,178.837,5.891,149.397
C08119=1157.686,-102.175,-42.800,178.839,5.891,149.396
C08120=1157.681,-101.903,-42.810,178.842,5.892,149.396
C08121=1157.676,-101.653,-42.819,178.844,5.892,149.395
C08122=1157.671,-101.404,-42.828,178.846,5.892,149.395
C08123=1157.665,-101.154,-42.838,178.848,5.893,149.394
C08124=1157.660,-100.904,-42.847,178.850,5.893,149.394
C08125=1157.655,-100.654,-42.856,178.852,5.893,149.393
C08126=1157.649,-100.405,-42.866,178.855,5.894,149.392
C08127=1157.644,-100.155,-42.875,178.856,5.894,149.392
C08128=1157.639,-99.905,-42.884,178.859,5.894,149.391
C08129=1157.633,-99.656,-42.894,178.861,5.895,149.391
C08130=1157.628,-99.406,-42.903,178.863,5.895,149.390
C08131=1157.622,-99.156,-42.912,178.865,5.895,149.390
C08132=1157.617,-98.906,-42.922,178.867,5.895,149.389
C08133=1157.612,-98.656,-42.931,178.869,5.896,149.389
C08134=1157.606,-98.407,-42.941,178.871,5.897,149.388
C08135=1157.601,-98.157,-42.950,178.873,5.896,149.387
C08136=1157.595,-97.907,-42.959,178.876,5.897,149.387
C08137=1157.591,-97.658,-42.969,178.877,5.897,149.386
C08138=1157.585,-97.408,-42.978,178.880,5.897,149.386
C08139=1157.579,-97.158,-42.987,178.882,5.898,149.385
C08140=1157.575,-96.908,-42.997,178.884,5.898,149.385
C08141=1157.569,-96.658,-43.007,178.886,5.899,149.384
C08142=1157.564,-96.408,-43.016,178.888,5.899,149.383
C08143=1157.559,-96.158,-43.026,178.890,5.899,149.383
C08144=1157.554,-95.909,-43.035,178.893,5.900,149.382
C08145=1157.549,-95.659,-43.044,178.894,5.900,149.382
C08146=1157.543,-95.409,-43.054,178.897,5.900,149.381
C08147=1157.538,-95.160,-43.063,178.899,5.901,149.381
C08148=1157.532,-94.910,-43.073,178.901,5.901,149.380
C08149=1157.527,-94.660,-43.083,178.903,5.902,149.380
C08150=1157.521,-94.410,-43.092,178.906,5.902,149.379
C08151=1157.516,-94.161,-43.102,178.907,5.902,149.378
C08152=1157.510,-93.911,-43.111,178.909,5.903,149.378
C08153=1157.505,-93.662,-43.121,178.912,5.902,149.377
C08154=1157.500,-93.411,-43.130,178.914,5.903,149.377
C08155=1157.495,-93.161,-43.140,178.916,5.904,149.376
C08156=1157.489,-92.911,-43.150,178.918,5.903,149.376
C08157=1157.485,-92.662,-43.159,178.920,5.904,149.375
C08158=1157.479,-92.412,-43.169,178.922,5.905,149.375
C08159=1157.474,-92.163,-43.178,178.924,5.905,149.374
C08160=1157.468,-91.912,-43.188,178.927,5.905,149.373
C08161=1157.463,-91.663,-43.198,178.928,5.905,149.373
C08162=1157.457,-91.413,-43.207,178.931,5.906,149.372
C08163=1157.452,-91.164,-43.217,178.933,5.906,149.372
C08164=1157.447,-90.914,-43.227,178.935,5.906,149.371
C08165=1157.442,-90.664,-43.236,178.937,5.907,149.371
C08166=1157.436,-90.414,-43.246,178.940,5.908,149.370
C08167=1157.431,-90.164,-43.255,178.941,5.908,149.370
C08168=1157.426,-89.915,-43.265,178.944,5.908,149.369
C08169=1157.420,-89.665,-43.275,178.946,5.909,149.368
C08170=1157.415,-89.415,-43.285,178.948,5.909,149.368
C08171=1157.410,-89.165,-43.295,178.950,5.909,149.367
C08172=1157.405,-88.915,-43.304,178.952,5.910,149.367
C08173=1157.399,-88.666,-43.314,178.955,5.909,149.366
C08174=1157.394,-88.417,-43.324,178.957,5.910,149.366
C08175=1157.388,-88.166,-43.333,178.958,5.910,149.365
C08176=1157.383,-87.917,-43.344,178.961,5.910,149.364
C08177=1157.378,-87.666,-43.353,178.963,5.911,149.364
C08178=1157.373,-87.417,-43.363,178.965,5.911,149.363
C08179=1157.368,-87.168,-43.373,178.967,5.912,149.363
C08180=1157.362,-86.917,-43.382,178.970,5.912,149.362
C08181=1157.356,-86.668,-43.392,178.971,5.912,149.362
C08182=1157.351,-86.419,-43.402,178.974,5.913,149.361
C08183=1157.346,-86.168,-43.413,178.976,5.914,149.360
C08184=1157.341,-85.918,-43.422,178.978,5.914,149.360
C08185=1157.336,-85.669,-43.432,178.980,5.914,149.359
C08186=1157.330,-85.419,-43.442,178.983,5.915,149.359
C08187=1157.325,-85.170,-43.451,178.985,5.914,149.358
C08188=1157.320,-84.919,-43.461,178.987,5.915,149.358
C08189=1157.314,-84.670,-43.472,178.989,5.916,149.357
C08190=1157.309,-84.421,-43.481,178.991,5.915,149.356
C08191=1157.304,-84.170,-43.491,178.993,5.916,149.356
C08192=1157.299,-83.920,-43.501,178.996,5.917,149.355
C08193=1157.294,-83.671,-43.511,178.998,5.917,149.355
C08194=1157.288,-83.421,-43.521,179.000,5.917,149.354
C08195=1157.282,-83.171,-43.531,179.002,5.918,149.354
C08196=1157.277,-82.922,-43.540,179.004,5.918,149.353
C08197=1157.272,-82.672,-43.551,179.006,5.918,149.353
C08198=1157.267,-82.422,-43.561,179.009,5.919,149.352
C08199=1157.261,-82.173,-43.571,179.011,5.920,149.351
C08200=1157.256,-81.923,-43.580,179.013,5.920,149.351
C08201=1157.251,-81.673,-43.591,179.015,5.920,149.350
C08202=1157.245,-81.423,-43.601,179.018,5.921,149.350
C08203=1157.241,-81.174,-43.610,179.020,5.920,149.349
C08204=1157.235,-80.924,-43.621,179.022,5.921,149.349
C08205=1157.230,-80.674,-43.631,179.024,5.922,149.348
C08206=1157.224,-80.424,-43.641,179.026,5.921,149.347
C08207=1157.219,-80.175,-43.650,179.028,5.922,149.347
C08208=1157.214,-79.925,-43.661,179.031,5.923,149.346
C08209=1157.209,-79.675,-43.671,179.033,5.923,149.346
C08210=1157.203,-79.425,-43.681,179.035,5.923,149.345
C08211=1157.198,-79.176,-43.691,179.037,5.924,149.344
C08212=1157.193,-78.926,-43.702,179.039,5.924,149.344
C08213=1157.188,-78.676,-43.712,179.041,5.925,149.344
C08214=1157.182,-78.427,-43.722,179.044,5.925,149.343
C08215=1157.176,-78.176,-43.731,179.046,5.926,149.342
C08216=1157.172,-77.927,-43.741,179.048,5.925,149.342
C08217=1157.166,-77.677,-43.752,179.050,5.926,149.341
C08218=1157.161,-77.427,-43.762,179.053,5.927,149.341
C08219=1157.156,-77.177,-43.772,179.055,5.926,149.340
C08220=1157.150,-76.928,-43.783,179.057,5.927,149.339
C08221=1157.145,-76.656,-43.794,179.059,5.928,149.339
C08222=1157.138,-76.385,-43.805,179.062,5.928,149.338
C08223=1157.133,-76.114,-43.816,179.064,5.929,149.338
C08224=1157.127,-75.843,-43.827,179.066,5.928,149.337
C08225=1157.122,-75.593,-43.837,179.069,5.929,149.336
C08226=1157.117,-75.344,-43.847,179.071,5.930,149.336
C08227=1157.112,-75.094,-43.858,179.073,5.930,149.335
C08228=1157.106,-74.844,-43.868,179.075,5.930,149.335
C08229=1157.100,-74.594,-43.878,179.078,5.931,149.334
C08230=1157.095,-74.344,-43.889,179.080,5.931,149.333
C08231=1157.090,-74.095,-43.899,179.082,5.931,149.333
C08232=1157.084,-73.845,-43.909,179.084,5.932,149.332
C08233=1157.079,-73.595,-43.920,179.086,5.933,149.332
C08234=1157.074,-73.345,-43.930,179.089,5.933,149.331
C08235=1157.069,-73.096,-43.939,179.091,5.933,149.331
C08236=1157.064,-72.846,-43.950,179.093,5.934,149.330
C08237=1157.058,-72.596,-43.960,179.096,5.934,149.329
C08238=1157.053,-72.346,-43.971,179.098,5.935,149.329
C08239=1157.048,-72.097,-43.981,179.100,5.934,149.328
C08240=1157.042,-71.847,-43.991,179.102,5.935,149.328
C08241=1157.037,-71.597,-44.002,179.105,5.936,149.327
C08242=1157.032,-71.348,-44.013,179.106,5.936,149.327
C08243=1157.026,-71.098,-44.023,179.108,5.936,149.326
C08244=1157.021,-70.848,-44.033,179.111,5.937,149.325
C08245=1157.016,-70.599,-44.044,179.113,5.938,149.325
C08246=1157.011,-70.348,-44.054,179.115,5.937,149.324
C08247=1157.005,-70.099,-44.064,179.118,5.938,149.324
C08248=1156.999,-69.849,-44.075,179.120,5.939,149.323
C08249=1156.995,-69.600,-44.086,179.122,5.939,149.323
C08250=1156.989,-69.350,-44.096,179.124,5.939,149.322
C08251=1156.984,-69.100,-44.107,179.127,5.939,149.321
C08252=1156.979,-68.851,-44.116,179.129,5.940,149.321
C08253=1156.974,-68.600,-44.127,179.132,5.941,149.320
C08254=1156.969,-68.351,-44.138,179.133,5.941,149.320
C08255=1156.963,-68.102,-44.148,179.135,5.941,149.319
C08256=1156.958,-67.852,-44.159,179.138,5.942,149.318
C08257=1156.953,-67.602,-44.169,179.140,5.943,149.318
C08258=1156.947,-67.351,-44.180,179.142,5.942,149.317
C08259=1156.942,-67.103,-44.191,179.144,5.943,149.317
C08260=1156.937,-66.852,-44.201,179.147,5.943,149.316
C08261=1156.931,-66.603,-44.212,179.149,5.944,149.316
C08262=1156.926,-66.353,-44.222,179.151,5.944,149.315
C08263=1156.921,-66.104,-44.233,179.154,5.945,149.314
C08264=1156.915,-65.854,-44.243,179.156,5.945,149.314
C08265=1156.910,-65.604,-44.254,179.158,5.946,149.313
C08266=1156.905,-65.354,-44.264,179.160,5.946,149.313
C08267=1156.900,-65.105,-44.275,179.163,5.946,149.312
C08268=1156.894,-64.855,-44.286,179.165,5.947,149.312
C08269=1156.889,-64.605,-44.296,179.167,5.948,149.311
C08270=1156.884,-64.356,-44.307,179.169,5.947,149.310
C08271=1156.879,-64.106,-44.318,179.171,5.948,149.310
C08272=1156.873,-63.856,-44.328,179.174,5.948,149.309
C08273=1156.869,-63.607,-44.339,179.176,5.949,149.309
C08274=1156.863,-63.357,-44.349,179.178,5.949,149.308
C08275=1156.858,-63.107,-44.360,179.180,5.950,149.308
C08276=1156.852,-62.857,-44.372,179.183,5.950,149.307
C08277=1156.847,-62.607,-44.382,179.185,5.951,149.306
C08278=1156.842,-62.358,-44.392,179.187,5.952,149.306
C08279=1156.837,-62.108,-44.404,179.190,5.951,149.305
C08280=1156.831,-61.859,-44.414,179.192,5.952,149.305
C08281=1156.827,-61.609,-44.425,179.194,5.952,149.304
C08282=1156.821,-61.359,-44.435,179.197,5.953,149.304
C08283=1156.816,-61.109,-44.446,179.199,5.953,149.303
C08284=1156.811,-60.859,-44.458,179.201,5.954,149.302
C08285=1156.805,-60.610,-44.468,179.203,5.954,149.302
C08286=1156.800,-60.360,-44.479,179.206,5.955,149.301
C08287=1156.795,-60.110,-44.490,179.208,5.956,149.301
C08288=1156.790,-59.860,-44.500,179.210,5.955,149.300
C08289=1156.784,-59.611,-44.511,179.212,5.956,149.300
C08290=1156.779,-59.361,-44.522,179.215,5.956,149.299
C08291=1156.773,-59.112,-44.533,179.217,5.957,149.298
C08292=1156.768,-58.862,-44.544,179.220,5.957,149.298
C08293=1156.764,-58.612,-44.555,179.221,5.957,149.297
C08294=1156.758,-58.362,-44.565,179.223,5.958,149.297
C08295=1156.753,-58.113,-44.576,179.226,5.959,149.296
C08296=1156.747,-57.863,-44.587,179.228,5.959,149.295
C08297=1156.742,-57.613,-44.599,179.230,5.959,149.295
C08298=1156.737,-57.363,-44.609,179.233,5.960,149.294
C08299=1156.732,-57.114,-44.620,179.235,5.960,149.294
C08300=1156.726,-56.864,-44.631,179.237,5.961,149.293
C08301=1156.721,-56.615,-44.642,179.240,5.961,149.292
C08302=1156.716,-56.364,-44.653,179.242,5.962,149.292
C08303=1156.711,-56.115,-44.664,179.244,5.962,149.291
C08304=1156.706,-55.866,-44.675,179.247,5.963,149.291
C08305=1156.700,-55.615,-44.686,179.249,5.963,149.290
C08306=1156.695,-55.366,-44.697,179.251,5.964,149.290
C08307=1156.690,-55.116,-44.708,179.254,5.965,149.289
C08308=1156.685,-54.867,-44.719,179.256,5.964,149.288
C08309=1156.679,-54.617,-44.730,179.258,5.965,149.288
C08310=1156.674,-54.367,-44.741,179.261,5.965,149.287
C08311=1156.670,-54.117,-44.752,179.263,5.966,149.287
C08312=1156.663,-53.868,-44.763,179.265,5.967,149.286
C08313=1156.659,-53.618,-44.774,179.267,5.967,149.286
C08314=1156.654,-53.368,-44.786,179.270,5.967,149.285
C08315=1156.648,-53.118,-44.796,179.272,5.968,149.284
C08316=1156.643,-52.869,-44.808,179.274,5.969,149.284
C08317=1156.638,-52.619,-44.819,179.277,5.969,149.283
C08318=1156.633,-52.370,-44.829,179.279,5.970,149.283
C08319=1156.627,-52.120,-44.841,179.281,5.969,149.282
C08320=1156.622,-51.870,-44.852,179.283,5.970,149.282
C08321=1156.617,-51.621,-44.863,179.286,5.971,149.281
C08322=1156.611,-51.371,-44.875,179.288,5.971,149.280
C08323=1156.607,-51.121,-44.886,179.291,5.972,149.280
C08324=1156.600,-50.871,-44.897,179.293,5.973,149.279
C08325=1156.596,-50.601,-44.909,179.296,5.973,149.278
C08326=1156.590,-50.331,-44.921,179.298,5.973,149.278
C08327=1156.584,-50.060,-44.933,179.300,5.974,149.277
C08328=1156.578,-49.789,-44.945,179.302,5.974,149.277
C08329=1156.573,-49.540,-44.956,179.305,5.975,149.276
C08330=1156.568,-49.290,-44.968,179.307,5.975,149.275
C08331=1156.563,-49.040,-44.979,179.309,5.976,149.275
C08332=1156.557,-48.790,-44.991,179.312,5.976,149.274
C08333=1156.552,-48.541,-45.002,179.314,5.977,149.274
C08334=1156.547,-48.291,-45.013,179.317,5.977,149.273
C08335=1156.541,-48.041,-45.024,179.319,5.977,149.273
C08336=1156.536,-47.792,-45.035,179.321,5.978,149.272
C08337=1156.531,-47.542,-45.047,179.323,5.979,149.271
C08338=1156.526,-47.292,-45.058,179.326,5.979,149.271
C08339=1156.521,-47.042,-45.070,179.328,5.980,149.270
C08340=1156.515,-46.793,-45.080,179.331,5.980,149.269
C08341=1156.510,-46.543,-45.092,179.333,5.981,149.269
C08342=1156.505,-46.293,-45.103,179.335,5.981,149.269
C08343=1156.500,-46.044,-45.115,179.337,5.981,149.268
C08344=1156.494,-45.794,-45.126,179.340,5.982,149.267
C08345=1156.489,-45.545,-45.138,179.342,5.983,149.267
C08346=1156.484,-45.295,-45.149,179.344,5.983,149.266
C08347=1156.479,-45.045,-45.161,179.347,5.984,149.265
C08348=1156.473,-44.795,-45.171,179.349,5.985,149.265
C08349=1156.468,-44.546,-45.183,179.351,5.984,149.264
C08350=1156.463,-44.296,-45.195,179.354,5.985,149.264
C08351=1156.458,-44.046,-45.206,179.356,5.985,149.263
C08352=1156.453,-43.796,-45.218,179.358,5.986,149.263
C08353=1156.447,-43.547,-45.229,179.361,5.987,149.262
C08354=1156.442,-43.297,-45.241,179.363,5.987,149.261
C08355=1156.437,-43.048,-45.252,179.366,5.988,149.261
C08356=1156.432,-42.798,-45.264,179.367,5.988,149.260
C08357=1156.427,-42.548,-45.275,179.370,5.988,149.260
C08358=1156.421,-42.299,-45.287,179.372,5.989,149.259
C08359=1156.416,-42.049,-45.299,179.375,5.989,149.258
C08360=1156.411,-41.799,-45.310,179.377,5.990,149.258
C08361=1156.406,-41.549,-45.322,179.380,5.991,149.257
C08362=1156.401,-41.300,-45.333,179.382,5.991,149.257
C08363=1156.395,-41.051,-45.344,179.385,5.992,149.256
C08364=1156.390,-40.801,-45.356,179.387,5.993,149.256
C08365=1156.385,-40.551,-45.368,179.389,5.992,149.255
C08366=1156.379,-40.301,-45.380,179.391,5.993,149.254
C08367=1156.375,-40.051,-45.391,179.393,5.994,149.254
C08368=1156.369,-39.801,-45.403,179.396,5.994,149.253
C08369=1156.364,-39.553,-45.414,179.398,5.995,149.253
C08370=1156.359,-39.303,-45.426,179.401,5.995,149.252
C08371=1156.353,-39.053,-45.437,179.403,5.996,149.252
C08372=1156.348,-38.803,-45.449,179.406,5.997,149.251
C08373=1156.343,-38.553,-45.461,179.408,5.997,149.250
C08374=1156.338,-38.303,-45.472,179.410,5.997,149.250
C08375=1156.333,-38.054,-45.484,179.412,5.998,149.249
C08376=1156.327,-37.804,-45.495,179.415,5.998,149.249
C08377=1156.322,-37.555,-45.507,179.417,5.999,149.248
C08378=1156.317,-37.305,-45.519,179.420,5.999,149.247
C08379=1156.312,-37.055,-45.531,179.422,6.000,149.247
C08380=1156.307,-36.806,-45.542,179.424,6.001,149.246
C08381=1156.301,-36.556,-45.554,179.427,6.001,149.246
C08382=1156.296,-36.306,-45.566,179.429,6.002,149.245
C08383=1156.291,-36.056,-45.578,179.432,6.003,149.245
C08384=1156.286,-35.808,-45.590,179.434,6.003,149.244
C08385=1156.280,-35.558,-45.602,179.436,6.003,149.243
C08386=1156.275,-35.308,-45.613,179.438,6.003,149.243
C08387=1156.270,-35.058,-45.625,179.441,6.004,149.242
C08388=1156.265,-34.808,-45.637,179.443,6.005,149.241
C08389=1156.260,-34.559,-45.649,179.445,6.006,149.241
C08390=1156.254,-34.309,-45.661,179.448,6.006,149.240
C08391=1156.249,-34.059,-45.672,179.450,6.007,149.240
C08392=1156.244,-33.809,-45.684,179.453,6.007,149.239
C08393=1156.239,-33.559,-45.696,179.455,6.008,149.239
C08394=1156.234,-33.310,-45.708,179.458,6.008,149.238
C08395=1156.229,-33.061,-45.720,179.460,6.009,149.238
C08396=1156.223,-32.811,-45.732,179.463,6.010,149.237
C08397=1156.218,-32.561,-45.744,179.465,6.010,149.236
C08398=1156.213,-32.312,-45.756,179.467,6.010,149.236
C08399=1156.207,-32.062,-45.767,179.469,6.011,149.235
C08400=1156.202,-31.812,-45.779,179.472,6.011,149.234
C08401=1156.197,-31.563,-45.792,179.474,6.012,149.234
C08402=1156.191,-31.313,-45.804,179.477,6.012,149.233
C08403=1156.187,-31.064,-45.815,179.479,6.013,149.233
C08404=1156.182,-30.814,-45.828,179.481,6.014,149.232
C08405=1156.176,-30.564,-45.839,179.484,6.014,149.232
C08406=1156.171,-30.314,-45.851,179.486,6.015,149.231
C08407=1156.166,-30.065,-45.864,179.488,6.016,149.230
C08408=1156.161,-29.815,-45.875,179.491,6.016,149.230
C08409=1156.156,-29.566,-45.887,179.493,6.017,149.229
C08410=1156.150,-29.316,-45.900,179.496,6.017,149.229
C08411=1156.145,-29.066,-45.912,179.498,6.018,149.228
C08412=1156.140,-28.816,-45.924,179.501,6.019,149.227
C08413=1156.134,-28.567,-45.936,179.503,6.019,149.227
C08414=1156.130,-28.317,-45.947,179.506,6.020,149.226
C08415=1156.125,-28.068,-45.960,179.508,6.021,149.226
C08416=1156.119,-27.818,-45.972,179.510,6.020,149.225
C08417=1156.114,-27.569,-45.984,179.512,6.021,149.225
C08418=1156.109,-27.319,-45.996,179.515,6.021,149.224
C08419=1156.103,-27.069,-46.008,179.517,6.022,149.223
C08420=1156.099,-26.819,-46.021,179.520,6.023,149.223
C08421=1156.093,-26.569,-46.033,179.522,6.023,149.222
C08422=1156.088,-26.320,-46.046,179.524,6.024,149.222
C08423=1156.083,-26.070,-46.057,179.527,6.025,149.221
C08424=1156.078,-25.821,-46.070,179.529,6.025,149.220
C08425=1156.073,-25.571,-46.081,179.531,6.026,149.220
C08426=1156.068,-25.321,-46.094,179.534,6.026,149.219
C08427=1156.062,-25.072,-46.106,179.536,6.027,149.219
C08428=1156.057,-24.822,-46.119,179.539,6.028,149.218
C08429=1156.052,-24.552,-46.132,179.541,6.028,149.218
C08430=1156.046,-24.283,-46.145,179.544,6.029,149.217
C08431=1156.040,-24.012,-46.158,179.546,6.029,149.216
C08432=1156.035,-23.742,-46.171,179.549,6.031,149.216
C08433=1156.030,-23.493,-46.184,179.552,6.031,149.215
C08434=1156.024,-23.243,-46.196,179.555,6.032,149.214
C08435=1156.019,-22.993,-46.208,179.557,6.032,149.214
C08436=1156.014,-22.744,-46.221,179.559,6.033,149.213
C08437=1156.009,-22.494,-46.233,179.562,6.034,149.213
C08438=1156.004,-22.245,-46.246,179.564,6.034,149.212
C08439=1155.998,-21.995,-46.257,179.566,6.034,149.212
C08440=1155.993,-21.745,-46.270,179.569,6.035,149.211
C08441=1155.988,-21.496,-46.283,179.571,6.035,149.210
C08442=1155.983,-21.245,-46.295,179.573,6.036,149.210
C08443=1155.978,-20.996,-46.307,179.576,6.037,149.209
C08444=1155.973,-20.747,-46.320,179.578,6.037,149.209
C08445=1155.967,-20.497,-46.332,179.580,6.038,149.208
C08446=1155.962,-20.248,-46.345,179.583,6.038,149.207
C08447=1155.957,-19.998,-46.357,179.585,6.039,149.207
C08448=1155.952,-19.748,-46.369,179.588,6.039,149.206
C08449=1155.947,-19.498,-46.382,179.590,6.040,149.206
C08450=1155.942,-19.249,-46.395,179.593,6.041,149.205
C08451=1155.936,-18.999,-46.407,179.595,6.042,149.205
C08452=1155.931,-18.749,-46.420,179.598,6.042,149.204
C08453=1155.926,-18.500,-46.432,179.600,6.043,149.203
C08454=1155.920,-18.250,-46.444,179.603,6.044,149.203
C08455=1155.915,-18.001,-46.457,179.605,6.045,149.202
C08456=1155.911,-17.751,-46.470,179.608,6.045,149.202
C08457=1155.905,-17.502,-46.482,179.610,6.046,149.201
C08458=1155.900,-17.252,-46.494,179.613,6.046,149.200
C08459=1155.895,-17.002,-46.507,179.615,6.047,149.200
C08460=1155.890,-16.753,-46.519,179.618,6.048,149.199
C08461=1155.885,-16.503,-46.533,179.620,6.049,149.199
C08462=1155.879,-16.253,-46.546,179.622,6.049,149.198
C08463=1155.874,-16.003,-46.558,179.625,6.050,149.198
C08464=1155.869,-15.754,-46.570,179.627,6.050,149.197
C08465=1155.864,-15.505,-46.583,179.629,6.051,149.196
C08466=1155.859,-15.255,-46.596,179.632,6.051,149.196
C08467=1155.854,-15.005,-46.608,179.634,6.052,149.195
C08468=1155.848,-14.755,-46.621,179.637,6.053,149.195
C08469=1155.843,-14.506,-46.633,179.639,6.053,149.194
C08470=1155.838,-14.256,-46.646,179.642,6.054,149.193
C08471=1155.833,-14.006,-46.659,179.644,6.055,149.193
C08472=1155.828,-13.757,-46.672,179.647,6.055,149.192
C08473=1155.822,-13.508,-46.685,179.649,6.056,149.192
C08474=1155.818,-13.258,-46.698,179.651,6.056,149.191
C08475=1155.813,-13.008,-46.710,179.654,6.057,149.191
C08476=1155.807,-12.759,-46.723,179.656,6.058,149.190
C08477=1155.802,-12.509,-46.735,179.658,6.058,149.189
C08478=1155.797,-12.259,-46.748,179.661,6.059,149.189
C08479=1155.792,-12.009,-46.761,179.663,6.060,149.188
C08480=1155.786,-11.760,-46.774,179.666,6.060,149.188
C08481=1155.781,-11.511,-46.786,179.668,6.061,149.187
C08482=1155.776,-11.260,-46.800,179.671,6.061,149.186
C08483=1155.771,-11.011,-46.812,179.673,6.062,149.186
C08484=1155.766,-10.762,-46.825,179.676,6.063,149.185
C08485=1155.761,-10.512,-46.838,179.678,6.064,149.185
C08486=1155.755,-10.262,-46.851,179.681,6.065,149.184
C08487=1155.750,-10.013,-46.864,179.683,6.065,149.184
C08488=1155.745,-9.763,-46.876,179.686,6.066,149.183
C08489=1155.741,-9.513,-46.889,179.688,6.067,149.183
C08490=1155.735,-9.264,-46.902,179.691,6.067,149.182
C08491=1155.730,-9.014,-46.915,179.693,6.068,149.181
C08492=1155.725,-8.764,-46.928,179.695,6.068,149.181
C08493=1155.719,-8.515,-46.941,179.698,6.069,149.180
C08494=1155.714,-8.266,-46.954,179.700,6.070,149.179
C08495=1155.710,-8.015,-46.967,179.702,6.070,149.179
C08496=1155.704,-7.766,-46.980,179.705,6.071,149.178
C08497=1155.699,-7.517,-46.993,179.707,6.072,149.178
C08498=1155.694,-7.267,-47.006,179.710,6.072,149.177
C08499=1155.689,-7.018,-47.019,179.713,6.073,149.176
C08500=1155.683,-6.768,-47.032,179.715,6.074,149.176
C08501=1155.679,-6.518,-47.045,179.718,6.075,149.175
C08502=1155.673,-6.269,-47.058,179.720,6.075,149.175
C08503=1155.669,-6.019,-47.071,179.723,6.076,149.174
C08504=1155.663,-5.769,-47.084,179.725,6.077,149.174
C08505=1155.658,-5.520,-47.097,179.728,6.077,149.173
C08506=1155.653,-5.270,-47.111,179.730,6.078,149.173
C08507=1155.648,-5.021,-47.124,179.733,6.078,149.172
C08508=1155.642,-4.771,-47.136,179.735,6.079,149.171
C08509=1155.638,-4.521,-47.149,179.737,6.080,149.171
C08510=1155.632,-4.272,-47.163,179.740,6.081,149.170
C08511=1155.628,-4.022,-47.176,179.743,6.082,149.170
C08512=1155.622,-3.773,-47.189,179.745,6.083,149.169
C08513=1155.617,-3.523,-47.202,179.748,6.083,149.168
C08514=1155.612,-3.273,-47.215,179.750,6.084,149.168
C08515=1155.606,-3.024,-47.228,179.752,6.084,149.167
C08516=1155.602,-2.774,-47.242,179.755,6.085,149.167
C08517=1155.596,-2.525,-47.255,179.757,6.086,149.166
C08518=1155.591,-2.275,-47.268,179.759,6.086,149.166
C08519=1155.586,-2.025,-47.281,179.762,6.087,149.165
C08520=1155.581,-1.776,-47.295,179.764,6.088,149.164
C08521=1155.576,-1.526,-47.308,179.768,6.089,149.164
C08522=1155.571,-1.277,-47.321,179.770,6.090,149.163
C08523=1155.566,-1.027,-47.335,179.772,6.090,149.163
C08524=1155.561,-0.778,-47.348,179.775,6.091,149.162
C08525=1155.555,-0.528,-47.361,179.777,6.091,149.161
C08526=1155.550,-0.278,-47.374,179.779,6.092,149.161
C08527=1155.545,-0.029,-47.388,179.782,6.093,149.160
C08528=1155.540,0.221,-47.401,179.784,6.093,149.160
C08529=1155.535,0.470,-47.415,179.787,6.094,149.159
C08530=1155.530,0.720,-47.428,179.790,6.096,149.159
C08531=1155.524,0.970,-47.441,179.792,6.096,149.158
C08532=1155.520,1.219,-47.454,179.794,6.097,149.158
C08533=1155.514,1.489,-47.468,179.797,6.097,149.157
C08534=1155.508,1.758,-47.483,179.800,6.098,149.156
C08535=1155.503,2.028,-47.498,179.803,6.099,149.156
C08536=1155.498,2.297,-47.512,179.805,6.100,149.155
C08537=1155.492,2.547,-47.525,179.808,6.100,149.154
C08538=1155.487,2.796,-47.539,179.810,6.101,149.154
C08539=1155.482,3.046,-47.552,179.813,6.101,149.153
C08540=1155.477,3.295,-47.566,179.815,6.103,149.153
C08541=1155.472,3.545,-47.579,179.818,6.103,149.152
C08542=1155.467,3.794,-47.593,179.820,6.104,149.152
C08543=1155.461,4.044,-47.606,179.823,6.105,149.151
C08544=1155.457,4.294,-47.620,179.825,6.106,149.150
C08545=1155.451,4.543,-47.633,179.828,6.106,149.150
C08546=1155.447,4.793,-47.647,179.830,6.107,149.149
C08547=1155.441,5.042,-47.660,179.833,6.108,149.149
C08548=1155.436,5.292,-47.674,179.835,6.109,149.148
C08549=1155.431,5.541,-47.687,179.838,6.109,149.147
C08550=1155.426,5.791,-47.701,179.840,6.110,149.147
C08551=1155.421,6.041,-47.715,179.843,6.111,149.146
C08552=1155.416,6.290,-47.728,179.845,6.111,149.146
C08553=1155.410,6.540,-47.742,179.848,6.112,149.145
C08554=1155.405,6.789,-47.756,179.850,6.114,149.145
C08555=1155.401,7.039,-47.769,179.853,6.114,149.144
C08556=1155.395,7.288,-47.783,179.855,6.115,149.144
C08557=1155.390,7.538,-47.797,179.858,6.115,149.143
C08558=1155.385,7.788,-47.810,179.860,6.116,149.142
C08559=1155.380,8.037,-47.824,179.863,6.117,149.142
C08560=1155.375,8.287,-47.838,179.866,6.118,149.141
C08561=1155.369,8.536,-47.851,179.868,6.119,149.141
C08562=1155.365,8.786,-47.865,179.870,6.119,149.140
C08563=1155.360,9.036,-47.878,179.873,6.120,149.139
C08564=1155.354,9.285,-47.892,179.875,6.121,149.139
C08565=1155.349,9.535,-47.907,179.878,6.121,149.138
C08566=1155.344,9.784,-47.919,179.881,6.123,149.138
C08567=1155.339,10.034,-47.934,179.883,6.123,149.137
C08568=1155.334,10.284,-47.948,179.885,6.124,149.137
C08569=1155.328,10.533,-47.961,179.888,6.125,149.136
C08570=1155.324,10.783,-47.975,179.890,6.125,149.136
C08571=1155.318,11.032,-47.989,179.893,6.127,149.135
C08572=1155.313,11.281,-48.003,179.896,6.127,149.134
C08573=1155.308,11.532,-48.016,179.898,6.128,149.134
C08574=1155.303,11.781,-48.030,179.900,6.129,149.133
C08575=1155.298,12.030,-48.044,179.903,6.129,149.133
C08576=1155.293,12.280,-48.058,179.906,6.131,149.132
C08577=1155.288,12.529,-48.071,179.909,6.131,149.131
C08578=1155.283,12.779,-48.086,179.911,6.132,149.131
C08579=1155.278,13.029,-48.100,179.913,6.133,149.130
C08580=1155.272,13.278,-48.114,179.916,6.133,149.130
C08581=1155.268,13.528,-48.127,179.919,6.135,149.129
C08582=1155.263,13.778,-48.141,179.921,6.135,149.129
C08583=1155.257,14.027,-48.155,179.924,6.136,149.128
C08584=1155.252,14.276,-48.169,179.926,6.137,149.128
C08585=1155.247,14.526,-48.184,179.928,6.137,149.127
C08586=1155.242,14.776,-48.198,179.931,6.139,149.126
C08587=1155.236,15.025,-48.211,179.934,6.139,149.126
C08588=1155.232,15.275,-48.225,179.936,6.140,149.125
C08589=1155.227,15.524,-48.239,179.939,6.141,149.125
C08590=1155.222,15.773,-48.253,179.941,6.141,149.124
C08591=1155.217,16.023,-48.267,179.944,6.143,149.123
C08592=1155.212,16.273,-48.282,179.946,6.143,149.123
C08593=1155.207,16.523,-48.296,179.949,6.144,149.122
C08594=1155.201,16.772,-48.310,179.951,6.145,149.122
C08595=1155.196,17.021,-48.324,179.954,6.145,149.121
C08596=1155.191,17.271,-48.338,179.956,6.147,149.121
C08597=1155.185,17.521,-48.351,179.959,6.147,149.120
C08598=1155.180,17.770,-48.366,179.961,6.148,149.120
C08599=1155.175,18.020,-48.380,179.964,6.149,149.119
C08600=1155.171,18.270,-48.394,179.967,6.150,149.118
C08601=1155.165,18.519,-48.408,179.969,6.151,149.118
C08602=1155.161,18.768,-48.422,179.972,6.151,149.117
C08603=1155.156,19.018,-48.436,179.974,6.152,149.117
C08604=1155.151,19.268,-48.450,179.977,6.154,149.116
C08605=1155.146,19.517,-48.465,179.980,6.154,149.115
C08606=1155.140,19.766,-48.479,179.982,6.155,149.115
C08607=1155.135,20.016,-48.493,179.984,6.155,149.114
C08608=1155.130,20.266,-48.507,179.987,6.157,149.114
C08609=1155.125,20.516,-48.522,179.990,6.157,149.113
C08610=1155.119,20.765,-48.536,179.992,6.158,149.113
C08611=1155.115,21.014,-48.551,179.995,6.159,149.112
C08612=1155.110,21.264,-48.565,179.997,6.160,149.112
C08613=1155.105,21.513,-48.580,180.000,6.161,149.111
C08614=1155.100,21.763,-48.594,-179.998,6.162,149.110
C08615=1155.095,22.013,-48.608,-179.996,6.162,149.110
C08616=1155.089,22.262,-48.622,-179.992,6.164,149.109
C08617=1155.084,22.511,-48.636,-179.990,6.165,149.109
C08618=1155.079,22.761,-48.651,-179.988,6.165,149.108
C08619=1155.074,23.011,-48.665,-179.985,6.166,149.108
C08620=1155.070,23.260,-48.680,-179.982,6.167,149.107
C08621=1155.065,23.510,-48.694,-179.980,6.168,149.107
C08622=1155.059,23.759,-48.708,-179.977,6.168,149.106
C08623=1155.054,24.008,-48.722,-179.975,6.169,149.105
C08624=1155.049,24.258,-48.737,-179.972,6.171,149.105
C08625=1155.044,24.508,-48.751,-179.970,6.171,149.104
C08626=1155.039,24.757,-48.766,-179.967,6.172,149.104
C08627=1155.034,25.007,-48.781,-179.965,6.173,149.103
C08628=1155.029,25.257,-48.795,-179.962,6.174,149.102
C08629=1155.023,25.506,-48.809,-179.960,6.175,149.102
C08630=1155.018,25.755,-48.823,-179.957,6.175,149.101
C08631=1155.014,26.004,-48.838,-179.954,6.177,149.101
C08632=1155.008,26.254,-48.853,-179.952,6.177,149.100
C08633=1155.003,26.504,-48.867,-179.949,6.178,149.100
C08634=1154.998,26.754,-48.882,-179.947,6.179,149.099
C08635=1154.994,27.003,-48.897,-179.944,6.180,149.099
C08636=1154.989,27.253,-48.911,-179.941,6.181,149.098
C08637=1154.983,27.522,-48.927,-179.939,6.182,149.098
C08638=1154.977,27.790,-48.943,-179.936,6.183,149.097
C08639=1154.972,28.059,-48.958,-179.933,6.183,149.096
C08640=1154.966,28.328,-48.974,-179.930,6.185,149.096
C08641=1154.961,28.577,-48.989,-179.928,6.185,149.095
C08642=1154.956,28.827,-49.003,-179.926,6.186,149.095
C08643=1154.951,29.077,-49.017,-179.922,6.187,149.094
C08644=1154.946,29.326,-49.032,-179.920,6.188,149.093
C08645=1154.941,29.576,-49.047,-179.918,6.189,149.093
C08646=1154.936,29.826,-49.061,-179.915,6.190,149.092
C08647=1154.931,30.075,-49.076,-179.912,6.191,149.092
C08648=1154.926,30.325,-49.091,-179.910,6.192,149.091
C08649=1154.921,30.574,-49.106,-179.907,6.193,149.090
C08650=1154.916,30.824,-49.121,-179.905,6.194,149.090
C08651=1154.911,31.073,-49.136,-179.902,6.194,149.089
C08652=1154.906,31.323,-49.150,-179.900,6.195,149.089
C08653=1154.901,31.572,-49.165,-179.897,6.197,149.088
C08654=1154.896,31.822,-49.180,-179.894,6.197,149.088
C08655=1154.891,32.071,-49.194,-179.892,6.198,149.087
C08656=1154.886,32.321,-49.210,-179.889,6.199,149.087
C08657=1154.881,32.570,-49.224,-179.887,6.200,149.086
C08658=1154.876,32.819,-49.239,-179.884,6.201,149.086
C08659=1154.870,33.069,-49.254,-179.881,6.202,149.085
C08660=1154.866,33.319,-49.269,-179.879,6.203,149.084
C08661=1154.861,33.568,-49.283,-179.877,6.204,149.084
C08662=1154.855,33.818,-49.299,-179.873,6.205,149.083
C08663=1154.850,34.067,-49.313,-179.871,6.206,149.083
C08664=1154.845,34.317,-49.328,-179.869,6.206,149.082
C08665=1154.840,34.566,-49.343,-179.866,6.208,149.082
C08666=1154.835,34.816,-49.358,-179.863,6.208,149.081
C08667=1154.830,35.065,-49.373,-179.861,6.209,149.081
C08668=1154.825,35.315,-49.388,-179.858,6.211,149.080
C08669=1154.820,35.564,-49.403,-179.856,6.211,149.079
C08670=1154.815,35.814,-49.417,-179.853,6.212,149.079
C08671=1154.810,36.063,-49.432,-179.850,6.213,149.078
C08672=1154.805,36.312,-49.448,-179.848,6.214,149.078
C08673=1154.800,36.562,-49.462,-179.845,6.215,149.077
C08674=1154.794,36.811,-49.478,-179.843,6.216,149.077
C08675=1154.789,37.061,-49.492,-179.840,6.217,149.076
C08676=1154.784,37.311,-49.508,-179.838,6.218,149.076
C08677=1154.779,37.560,-49.523,-179.835,6.219,149.075
C08678=1154.774,37.809,-49.537,-179.832,6.220,149.075
C08679=1154.770,38.059,-49.553,-179.829,6.221,149.074
C08680=1154.765,38.309,-49.568,-179.827,6.222,149.073
C08681=1154.760,38.558,-49.584,-179.825,6.223,149.073
C08682=1154.755,38.808,-49.598,-179.822,6.224,149.072
C08683=1154.749,39.057,-49.613,-179.820,6.225,149.072
C08684=1154.745,39.306,-49.628,-179.817,6.225,149.071
C08685=1154.739,39.556,-49.643,-179.814,6.227,149.071
C08686=1154.734,39.805,-49.658,-179.811,6.227,149.070
C08687=1154.729,40.055,-49.674,-179.809,6.228,149.070
C08688=1154.725,40.304,-49.689,-179.806,6.230,149.069
C08689=1154.719,40.554,-49.704,-179.804,6.230,149.068
C08690=1154.714,40.804,-49.720,-179.801,6.232,149.068
C08691=1154.709,41.053,-49.735,-179.799,6.233,149.067
C08692=1154.704,41.302,-49.750,-179.796,6.233,149.067
C08693=1154.699,41.551,-49.765,-179.793,6.235,149.066
C08694=1154.693,41.801,-49.780,-179.791,6.236,149.066
C08695=1154.689,42.051,-49.796,-179.788,6.237,149.065
C08696=1154.684,42.301,-49.811,-179.786,6.238,149.065
C08697=1154.679,42.550,-49.826,-179.783,6.238,149.064
C08698=1154.674,42.799,-49.842,-179.780,6.240,149.064
C08699=1154.668,43.049,-49.857,-179.778,6.240,149.063
C08700=1154.664,43.298,-49.872,-179.775,6.241,149.062
C08701=1154.659,43.548,-49.888,-179.773,6.243,149.062
C08702=1154.654,43.797,-49.903,-179.770,6.243,149.061
C08703=1154.649,44.047,-49.918,-179.767,6.245,149.061
C08704=1154.643,44.296,-49.934,-179.765,6.245,149.060
C08705=1154.639,44.545,-49.949,-179.762,6.246,149.060
C08706=1154.634,44.795,-49.965,-179.759,6.248,149.059
C08707=1154.628,45.045,-49.980,-179.757,6.248,149.059
C08708=1154.624,45.294,-49.995,-179.754,6.250,149.058
C08709=1154.618,45.543,-50.011,-179.752,6.250,149.058
C08710=1154.613,45.793,-50.026,-179.750,6.251,149.057
C08711=1154.609,46.043,-50.042,-179.746,6.253,149.056
C08712=1154.604,46.292,-50.057,-179.744,6.253,149.056
C08713=1154.598,46.541,-50.073,-179.741,6.255,149.055
C08714=1154.594,46.790,-50.088,-179.739,6.256,149.055
C08715=1154.589,47.041,-50.104,-179.735,6.257,149.054
C08716=1154.583,47.290,-50.119,-179.733,6.258,149.054
C08717=1154.579,47.539,-50.134,-179.731,6.259,149.053
C08718=1154.573,47.788,-50.150,-179.728,6.260,149.053
C08719=1154.569,48.039,-50.166,-179.726,6.261,149.052
C08720=1154.563,48.288,-50.182,-179.723,6.262,149.051
C08721=1154.559,48.537,-50.197,-179.720,6.263,149.051
C08722=1154.553,48.786,-50.212,-179.718,6.263,149.050
C08723=1154.548,49.037,-50.228,-179.715,6.265,149.050
C08724=1154.543,49.286,-50.244,-179.713,6.266,149.049
C08725=1154.539,49.534,-50.259,-179.710,6.267,149.049
C08726=1154.534,49.785,-50.275,-179.707,6.268,149.048
C08727=1154.528,50.034,-50.291,-179.704,6.269,149.048
C08728=1154.523,50.283,-50.307,-179.702,6.270,149.047
C08729=1154.518,50.532,-50.322,-179.699,6.271,149.047
C08730=1154.514,50.783,-50.337,-179.697,6.272,149.046
C08731=1154.508,51.032,-50.353,-179.695,6.273,149.046
C08732=1154.503,51.281,-50.369,-179.691,6.274,149.045
C08733=1154.498,51.531,-50.385,-179.689,6.275,149.045
C08734=1154.494,51.780,-50.400,-179.686,6.277,149.044
C08735=1154.488,52.029,-50.416,-179.684,6.277,149.044
C08736=1154.484,52.279,-50.432,-179.681,6.279,149.043
C08737=1154.479,52.528,-50.448,-179.678,6.280,149.042
C08738=1154.473,52.778,-50.464,-179.676,6.281,149.042
C08739=1154.468,53.028,-50.480,-179.673,6.282,149.041
C08740=1154.464,53.277,-50.495,-179.671,6.283,149.041
C08741=1154.458,53.545,-50.512,-179.668,6.284,149.040
C08742=1154.453,53.814,-50.529,-179.665,6.285,149.040
C08743=1154.448,54.083,-50.546,-179.662,6.286,149.039
C08744=1154.442,54.351,-50.563,-179.659,6.287,149.038
C08745=1154.437,54.600,-50.579,-179.656,6.289,149.038
C08746=1154.432,54.850,-50.595,-179.654,6.289,149.037
C08747=1154.427,55.100,-50.611,-179.651,6.290,149.037
C08748=1154.422,55.348,-50.627,-179.649,6.292,149.036
C08749=1154.417,55.599,-50.643,-179.646,6.292,149.036
C08750=1154.412,55.848,-50.659,-179.643,6.294,149.035
C08751=1154.407,56.097,-50.676,-179.641,6.295,149.035
C08752=1154.402,56.347,-50.691,-179.638,6.296,149.034
C08753=1154.397,56.596,-50.707,-179.636,6.297,149.034
C08754=1154.392,56.846,-50.723,-179.633,6.298,149.033
C08755=1154.386,57.095,-50.739,-179.630,6.299,149.033
C08756=1154.383,57.344,-50.755,-179.627,6.300,149.032
C08757=1154.377,57.594,-50.771,-179.625,6.301,149.032
C08758=1154.373,57.843,-50.787,-179.622,6.303,149.031
C08759=1154.367,58.093,-50.803,-179.620,6.304,149.030
C08760=1154.362,58.342,-50.818,-179.617,6.305,149.030
C08761=1154.358,58.592,-50.835,-179.614,6.306,149.029
C08762=1154.352,58.841,-50.851,-179.611,6.307,149.029
C08763=1154.348,59.090,-50.867,-179.609,6.308,149.028
C08764=1154.342,59.340,-50.884,-179.606,6.309,149.028
C08765=1154.337,59.590,-50.900,-179.604,6.310,149.027
C08766=1154.332,59.839,-50.916,-179.601,6.312,149.027
C08767=1154.327,60.088,-50.932,-179.599,6.312,149.026
C08768=1154.322,60.338,-50.948,-179.596,6.314,149.026
C08769=1154.317,60.587,-50.965,-179.593,6.315,149.025
C08770=1154.312,60.836,-50.981,-179.590,6.316,149.025
C08771=1154.307,61.086,-50.997,-179.588,6.317,149.024
C08772=1154.302,61.335,-51.013,-179.585,6.318,149.024
C08773=1154.298,61.585,-51.029,-179.583,6.319,149.023
C08774=1154.293,61.834,-51.046,-179.580,6.321,149.023
C08775=1154.288,62.084,-51.062,-179.578,6.321,149.022
C08776=1154.283,62.333,-51.078,-179.574,6.323,149.021
C08777=1154.278,62.582,-51.094,-179.572,6.324,149.021
C08778=1154.272,62.832,-51.111,-179.569,6.325,149.021
C08779=1154.268,63.082,-51.127,-179.567,6.326,149.020
C08780=1154.262,63.331,-51.143,-179.564,6.327,149.019
C08781=1154.258,63.580,-51.160,-179.561,6.329,149.019
C08782=1154.253,63.829,-51.176,-179.559,6.330,149.018
C08783=1154.248,64.079,-51.192,-179.556,6.331,149.018
C08784=1154.243,64.328,-51.208,-179.553,6.332,149.017
C08785=1154.238,64.578,-51.225,-179.551,6.333,149.017
C08786=1154.232,64.827,-51.242,-179.548,6.334,149.016
C08787=1154.228,65.077,-51.258,-179.545,6.336,149.016
C08788=1154.223,65.326,-51.274,-179.543,6.336,149.015
C08789=1154.218,65.575,-51.291,-179.540,6.338,149.015
C08790=1154.213,65.825,-51.307,-179.538,6.339,149.014
C08791=1154.208,66.074,-51.323,-179.535,6.340,149.014
C08792=1154.203,66.324,-51.340,-179.532,6.341,149.013
C08793=1154.199,66.573,-51.357,-179.529,6.342,149.013
C08794=1154.193,66.822,-51.373,-179.527,6.344,149.012
C08795=1154.188,67.072,-51.390,-179.524,6.345,149.012
C08796=1154.183,67.321,-51.406,-179.521,6.346,149.011
C08797=1154.178,67.571,-51.423,-179.519,6.347,149.010
C08798=1154.174,67.820,-51.439,-179.516,6.348,149.010
C08799=1154.169,68.069,-51.456,-179.514,6.349,149.010
C08800=1154.163,68.319,-51.472,-179.511,6.351,149.009
C08801=1154.158,68.568,-51.488,-179.508,6.351,149.009
C08802=1154.154,68.818,-51.505,-179.506,6.353,149.008
C08803=1154.149,69.067,-51.522,-179.503,6.354,149.007
C08804=1154.143,69.316,-51.539,-179.500,6.355,149.007
C08805=1154.139,69.566,-51.555,-179.498,6.357,149.007
C08806=1154.135,69.815,-51.572,-179.495,6.357,149.006
C08807=1154.129,70.064,-51.589,-179.492,6.359,149.005
C08808=1154.124,70.314,-51.605,-179.490,6.360,149.005
C08809=1154.119,70.564,-51.622,-179.487,6.361,149.004
C08810=1154.114,70.813,-51.638,-179.484,6.363,149.004
C08811=1154.109,71.062,-51.655,-179.482,6.363,149.003
C08812=1154.105,71.312,-51.672,-179.479,6.365,149.003
C08813=1154.099,71.561,-51.689,-179.477,6.366,149.002
C08814=1154.094,71.810,-51.705,-179.473,6.367,149.002
C08815=1154.089,72.060,-51.723,-179.471,6.369,149.001
C08816=1154.084,72.309,-51.739,-179.469,6.370,149.001
C08817=1154.080,72.559,-51.756,-179.465,6.371,149.000
C08818=1154.074,72.808,-51.773,-179.463,6.372,149.000
C08819=1154.069,73.057,-51.789,-179.460,6.374,148.999
C08820=1154.064,73.307,-51.806,-179.458,6.374,148.999
C08821=1154.060,73.556,-51.823,-179.455,6.376,148.998
C08822=1154.055,73.806,-51.840,-179.452,6.377,148.998
C08823=1154.049,74.055,-51.857,-179.450,6.378,148.997
C08824=1154.045,74.304,-51.874,-179.447,6.380,148.997
C08825=1154.040,74.554,-51.891,-179.444,6.380,148.996
C08826=1154.035,74.803,-51.908,-179.442,6.382,148.996
C08827=1154.030,75.052,-51.925,-179.439,6.384,148.995
C08828=1154.025,75.302,-51.942,-179.436,6.384,148.995
C08829=1154.021,75.551,-51.958,-179.433,6.386,148.994
C08830=1154.015,75.801,-51.976,-179.431,6.387,148.994
C08831=1154.010,76.050,-51.992,-179.428,6.388,148.993
C08832=1154.005,76.300,-52.009,-179.425,6.390,148.993
C08833=1154.001,76.548,-52.026,-179.423,6.390,148.992
C08834=1153.996,76.798,-52.044,-179.420,6.392,148.992
C08835=1153.991,77.047,-52.060,-179.417,6.393,148.991
C08836=1153.985,77.297,-52.077,-179.415,6.394,148.991
C08837=1153.981,77.546,-52.094,-179.412,6.396,148.990
C08838=1153.976,77.795,-52.112,-179.410,6.397,148.990
C08839=1153.970,78.045,-52.129,-179.407,6.398,148.989
C08840=1153.966,78.294,-52.146,-179.404,6.399,148.989
C08841=1153.960,78.544,-52.163,-179.402,6.400,148.988
C08842=1153.956,78.793,-52.180,-179.399,6.402,148.988
C08843=1153.951,79.042,-52.197,-179.396,6.403,148.987
C08844=1153.947,79.292,-52.214,-179.394,6.404,148.987
C08845=1153.941,79.560,-52.232,-179.391,6.406,148.986
C08846=1153.935,79.829,-52.251,-179.388,6.407,148.986
C08847=1153.930,80.096,-52.270,-179.385,6.409,148.985
C08848=1153.925,80.365,-52.288,-179.382,6.410,148.985
C08849=1153.920,80.615,-52.306,-179.379,6.411,148.984
C08850=1153.915,80.864,-52.322,-179.376,6.412,148.983
C08851=1153.910,81.114,-52.340,-179.373,6.414,148.983
C08852=1153.905,81.362,-52.356,-179.371,6.415,148.983
C08853=1153.900,81.612,-52.374,-179.368,6.416,148.982
C08854=1153.895,81.861,-52.392,-179.365,6.418,148.981
C08855=1153.891,82.111,-52.408,-179.363,6.419,148.981
C08856=1153.886,82.360,-52.426,-179.360,6.420,148.980
C08857=1153.880,82.610,-52.444,-179.357,6.422,148.980
C08858=1153.876,82.859,-52.461,-179.355,6.423,148.980
C08859=1153.871,83.108,-52.478,-179.352,6.424,148.979
C08860=1153.865,83.358,-52.495,-179.349,6.426,148.978
C08861=1153.861,83.606,-52.513,-179.347,6.427,148.978
C08862=1153.856,83.856,-52.530,-179.344,6.428,148.978
C08863=1153.851,84.105,-52.548,-179.341,6.430,148.977
C08864=1153.846,84.355,-52.564,-179.339,6.430,148.977
C08865=1153.842,84.604,-52.582,-179.336,6.432,148.976
C08866=1153.836,84.854,-52.600,-179.333,6.433,148.975
C08867=1153.831,85.103,-52.618,-179.331,6.434,148.975
C08868=1153.827,85.352,-52.634,-179.328,6.436,148.975
C08869=1153.822,85.602,-52.652,-179.325,6.438,148.974
C08870=1153.817,85.851,-52.670,-179.323,6.438,148.974
C08871=1153.812,86.101,-52.688,-179.320,6.440,148.973
C08872=1153.807,86.350,-52.704,-179.317,6.442,148.973
C08873=1153.803,86.599,-52.722,-179.315,6.442,148.972
C08874=1153.797,86.848,-52.740,-179.312,6.444,148.972
C08875=1153.792,87.098,-52.757,-179.309,6.445,148.971
C08876=1153.787,87.347,-52.775,-179.307,6.446,148.971
C08877=1153.782,87.596,-52.792,-179.304,6.448,148.970
C08878=1153.777,87.845,-52.810,-179.301,6.449,148.970
C08879=1153.773,88.095,-52.828,-179.298,6.451,148.969
C08880=1153.767,88.344,-52.845,-179.296,6.451,148.969
C08881=1153.762,88.594,-52.863,-179.293,6.453,148.968
C08882=1153.758,88.843,-52.881,-179.290,6.455,148.968
C08883=1153.753,89.092,-52.898,-179.288,6.455,148.967
C08884=1153.748,89.341,-52.916,-179.285,6.457,148.967
C08885=1153.743,89.591,-52.934,-179.282,6.459,148.966
C08886=1153.738,89.840,-52.951,-179.279,6.460,148.966
C08887=1153.733,90.090,-52.969,-179.277,6.461,148.965
C08888=1153.728,90.339,-52.987,-179.274,6.463,148.965
C08889=1153.723,90.588,-53.005,-179.271,6.464,148.964
C08890=1153.719,90.837,-53.021,-179.269,6.465,148.964
C08891=1153.714,91.087,-53.039,-179.266,6.466,148.963
C08892=1153.709,91.336,-53.057,-179.263,6.468,148.963
C08893=1153.705,91.586,-53.076,-179.261,6.470,148.963
C08894=1153.699,91.835,-53.093,-179.258,6.470,148.962
C08895=1153.695,92.085,-53.111,-179.255,6.472,148.961
C08896=1153.690,92.334,-53.129,-179.252,6.474,148.961
C08897=1153.685,92.583,-53.147,-179.250,6.475,148.961
C08898=1153.680,92.832,-53.165,-179.247,6.476,148.960
C08899=1153.675,93.081,-53.183,-179.244,6.478,148.960
C08900=1153.670,93.331,-53.200,-179.242,6.479,148.959
C08901=1153.665,93.580,-53.218,-179.240,6.480,148.959
C08902=1153.660,93.829,-53.236,-179.236,6.482,148.958
C08903=1153.655,94.079,-53.254,-179.234,6.483,148.958
C08904=1153.650,94.328,-53.272,-179.231,6.485,148.957
C08905=1153.645,94.577,-53.290,-179.229,6.486,148.957
C08906=1153.641,94.827,-53.308,-179.226,6.487,148.956
C08907=1153.636,95.076,-53.326,-179.223,6.489,148.956
C08908=1153.631,95.325,-53.344,-179.220,6.490,148.955
C08909=1153.626,95.574,-53.362,-179.217,6.491,148.955
C08910=1153.621,95.824,-53.380,-179.215,6.493,148.954
C08911=1153.616,96.073,-53.398,-179.212,6.494,148.954
C08912=1153.611,96.322,-53.416,-179.209,6.496,148.953
C08913=1153.606,96.572,-53.434,-179.207,6.497,148.953
C08914=1153.602,96.822,-53.452,-179.204,6.498,148.952
C08915=1153.597,97.071,-53.470,-179.201,6.500,148.952
C08916=1153.592,97.320,-53.488,-179.198,6.502,148.952
C08917=1153.587,97.569,-53.506,-179.196,6.503,148.951
C08918=1153.582,97.818,-53.524,-179.193,6.504,148.950
C08919=1153.577,98.067,-53.543,-179.190,6.506,148.950
C08920=1153.572,98.316,-53.561,-179.188,6.507,148.950
C08921=1153.568,98.566,-53.579,-179.185,6.509,148.949
C08922=1153.563,98.815,-53.597,-179.182,6.509,148.949
C08923=1153.558,99.064,-53.615,-179.180,6.511,148.948
C08924=1153.553,99.314,-53.633,-179.177,6.513,148.948
C08925=1153.548,99.563,-53.651,-179.174,6.515,148.947
C08926=1153.544,99.813,-53.670,-179.171,6.515,148.947
C08927=1153.538,100.062,-53.688,-179.169,6.517,148.946
C08928=1153.533,100.311,-53.706,-179.166,6.518,148.946
C08929=1153.528,100.560,-53.725,-179.163,6.520,148.945
C08930=1153.524,100.809,-53.743,-179.160,6.521,148.945
C08931=1153.519,101.059,-53.761,-179.158,6.522,148.944
C08932=1153.514,101.308,-53.779,-179.155,6.524,148.944
C08933=1153.509,101.558,-53.798,-179.152,6.526,148.944
C08934=1153.504,101.807,-53.816,-179.150,6.527,148.943
C08935=1153.500,102.056,-53.835,-179.147,6.529,148.943
C08936=1153.495,102.305,-53.853,-179.144,6.530,148.942
C08937=1153.489,102.555,-53.871,-179.142,6.531,148.942
C08938=1153.484,102.804,-53.889,-179.139,6.533,148.941
C08939=1153.480,103.053,-53.908,-179.136,6.534,148.941
C08940=1153.475,103.302,-53.926,-179.133,6.536,148.940
C08941=1153.470,103.552,-53.945,-179.131,6.537,148.940
C08942=1153.465,103.801,-53.963,-179.128,6.539,148.939
C08943=1153.461,104.050,-53.982,-179.125,6.540,148.939
C08944=1153.456,104.299,-54.000,-179.122,6.542,148.938
C08945=1153.450,104.549,-54.019,-179.119,6.543,148.938
C08946=1153.446,104.798,-54.038,-179.117,6.545,148.938
C08947=1153.441,105.047,-54.056,-179.115,6.546,148.937
C08948=1153.436,105.297,-54.074,-179.112,6.548,148.937
C08949=1153.431,105.564,-54.094,-179.109,6.549,148.936
C08950=1153.426,105.834,-54.115,-179.106,6.551,148.936
C08951=1153.421,106.102,-54.134,-179.103,6.552,148.935
C08952=1153.415,106.370,-54.155,-179.100,6.554,148.935
C08953=1153.410,106.619,-54.173,-179.097,6.555,148.934
C08954=1153.406,106.869,-54.191,-179.095,6.557,148.934
C08955=1153.401,107.118,-54.211,-179.092,6.559,148.933
C08956=1153.396,107.367,-54.228,-179.089,6.560,148.933
C08957=1153.392,107.616,-54.248,-179.086,6.562,148.932
C08958=1153.386,107.866,-54.266,-179.084,6.563,148.932
C08959=1153.381,108.114,-54.285,-179.081,6.564,148.932
C08960=1153.376,108.365,-54.304,-179.078,6.566,148.931
C08961=1153.372,108.613,-54.322,-179.075,6.567,148.930
C08962=1153.367,108.863,-54.341,-179.072,6.569,148.930
C08963=1153.362,109.112,-54.360,-179.070,6.571,148.930
C08964=1153.357,109.361,-54.378,-179.067,6.573,148.929
C08965=1153.352,109.611,-54.398,-179.065,6.573,148.929
C08966=1153.347,109.860,-54.416,-179.062,6.575,148.928
C08967=1153.342,110.109,-54.435,-179.059,6.576,148.928
C08968=1153.338,110.359,-54.453,-179.056,6.578,148.927
C08969=1153.333,110.607,-54.472,-179.053,6.580,148.927
C08970=1153.328,110.857,-54.492,-179.051,6.582,148.927
C08971=1153.324,111.106,-54.510,-179.048,6.583,148.926
C08972=1153.318,111.355,-54.529,-179.045,6.584,148.926
C08973=1153.314,111.605,-54.547,-179.043,6.585,148.925
C08974=1153.309,111.853,-54.567,-179.040,6.587,148.925
C08975=1153.305,112.103,-54.586,-179.037,6.589,148.924
C08976=1153.299,112.352,-54.604,-179.035,6.591,148.924
C08977=1153.295,112.601,-54.623,-179.032,6.592,148.924
C08978=1153.290,112.850,-54.643,-179.029,6.594,148.923
C08979=1153.284,113.100,-54.661,-179.026,6.595,148.922
C08980=1153.280,113.349,-54.680,-179.024,6.596,148.922
C08981=1153.275,113.598,-54.700,-179.021,6.598,148.922
C08982=1153.270,113.848,-54.718,-179.018,6.600,148.921
C08983=1153.265,114.097,-54.737,-179.016,6.601,148.921
C08984=1153.261,114.346,-54.756,-179.013,6.603,148.920
C08985=1153.256,114.595,-54.775,-179.010,6.604,148.920
C08986=1153.250,114.845,-54.794,-179.007,6.606,148.919
C08987=1153.246,115.094,-54.813,-179.004,6.608,148.919
C08988=1153.241,115.343,-54.833,-179.001,6.609,148.919
C08989=1153.237,115.592,-54.851,-178.999,6.610,148.918
C08990=1153.232,115.841,-54.871,-178.997,6.612,148.918
C08991=1153.226,116.091,-54.890,-178.994,6.614,148.917
C08992=1153.222,116.340,-54.909,-178.991,6.615,148.917
C08993=1153.217,116.589,-54.928,-178.988,6.617,148.916
C08994=1153.212,116.838,-54.948,-178.985,6.618,148.916
C08995=1153.207,117.087,-54.966,-178.983,6.620,148.916
C08996=1153.203,117.337,-54.986,-178.980,6.622,148.915
C08997=1153.197,117.586,-55.005,-178.977,6.624,148.915
C08998=1153.193,117.835,-55.024,-178.974,6.625,148.914
C08999=1153.188,118.084,-55.043,-178.971,6.627,148.914
C09000=1153.183,118.334,-55.063,-178.969,6.628,148.913
C09001=1153.178,118.582,-55.081,-178.966,6.629,148.913
C09002=1153.174,118.832,-55.101,-178.964,6.631,148.912
C09003=1153.169,119.081,-55.121,-178.961,6.633,148.912
C09004=1153.164,119.330,-55.140,-178.958,6.634,148.912
C09005=1153.160,119.580,-55.159,-178.955,6.636,148.911
C09006=1153.154,119.828,-55.178,-178.953,6.638,148.911
C09007=1153.149,120.078,-55.198,-178.950,6.639,148.910
C09008=1153.145,120.328,-55.218,-178.947,6.641,148.910
C09009=1153.140,120.576,-55.236,-178.944,6.643,148.909
C09010=1153.135,120.826,-55.256,-178.941,6.644,148.909
C09011=1153.130,121.074,-55.275,-178.939,6.646,148.909
C09012=1153.125,121.324,-55.295,-178.936,6.648,148.908
C09013=1153.121,121.573,-55.314,-178.933,6.649,148.908
C09014=1153.116,121.822,-55.333,-178.931,6.651,148.907
C09015=1153.111,122.072,-55.353,-178.928,6.653,148.907
C09016=1153.106,122.321,-55.372,-178.925,6.653,148.906
C09017=1153.101,122.570,-55.392,-178.922,6.655,148.906
C09018=1153.097,122.819,-55.411,-178.920,6.657,148.906
C09019=1153.092,123.068,-55.431,-178.917,6.658,148.905
C09020=1153.087,123.317,-55.451,-178.914,6.660,148.905
C09021=1153.083,123.567,-55.470,-178.912,6.662,148.904
C09022=1153.077,123.816,-55.490,-178.909,6.664,148.904
C09023=1153.072,124.065,-55.509,-178.906,6.665,148.904
C09024=1153.068,124.315,-55.529,-178.903,6.667,148.903
C09025=1153.063,124.563,-55.548,-178.901,6.669,148.903
C09026=1153.059,124.812,-55.568,-178.898,6.670,148.902
C09027=1153.054,125.062,-55.588,-178.895,6.672,148.902
C09028=1153.049,125.311,-55.607,-178.892,6.673,148.901
C09029=1153.044,125.560,-55.627,-178.889,6.675,148.901
C09030=1153.039,125.809,-55.647,-178.887,6.677,148.901
C09031=1153.034,126.058,-55.666,-178.884,6.679,148.900
C09032=1153.029,126.308,-55.686,-178.881,6.680,148.900
C09033=1153.025,126.557,-55.706,-178.879,6.682,148.899
C09034=1153.020,126.806,-55.726,-178.876,6.684,148.899
C09035=1153.015,127.055,-55.745,-178.873,6.685,148.899
C09036=1153.010,127.305,-55.765,-178.870,6.687,148.898
C09037=1153.006,127.553,-55.785,-178.868,6.689,148.898
C09038=1153.001,127.802,-55.804,-178.864,6.690,148.897
C09039=1152.996,128.052,-55.824,-178.862,6.692,148.897
C09040=1152.992,128.301,-55.844,-178.859,6.694,148.896
C09041=1152.987,128.550,-55.864,-178.856,6.695,148.896
C09042=1152.982,128.799,-55.883,-178.854,6.697,148.896
C09043=1152.977,129.048,-55.903,-178.851,6.699,148.895
C09044=1152.973,129.298,-55.923,-178.848,6.700,148.895
C09045=1152.967,129.547,-55.944,-178.845,6.702,148.894
C09046=1152.962,129.796,-55.963,-178.843,6.704,148.894
C09047=1152.957,130.045,-55.983,-178.840,6.706,148.894
C09048=1152.953,130.294,-56.003,-178.837,6.707,148.893
C09049=1152.948,130.544,-56.023,-178.835,6.709,148.893
C09050=1152.944,130.793,-56.043,-178.832,6.711,148.892
C09051=1152.938,131.042,-56.062,-178.829,6.712,148.892
C09052=1152.934,131.291,-56.083,-178.826,6.714,148.892
C09053=1152.929,131.559,-56.104,-178.823,6.716,148.891
C09054=1152.923,131.828,-56.126,-178.821,6.717,148.891
C09055=1152.919,132.096,-56.147,-178.817,6.720,148.890
C09056=1152.913,132.365,-56.169,-178.815,6.721,148.890
C09057=1152.908,132.615,-56.189,-178.812,6.723,148.889
C09058=1152.904,132.864,-56.209,-178.809,6.725,148.889
C09059=1152.899,133.113,-56.230,-178.806,6.727,148.889
C09060=1152.894,133.362,-56.249,-178.804,6.728,148.888
C09061=1152.890,133.611,-56.269,-178.801,6.730,148.888
C09062=1152.884,133.860,-56.289,-178.798,6.732,148.888
C09063=1152.880,134.109,-56.310,-178.796,6.733,148.887
C09064=1152.875,134.358,-56.330,-178.793,6.735,148.887
C09065=1152.871,134.608,-56.350,-178.790,6.737,148.886
C09066=1152.866,134.857,-56.370,-178.787,6.738,148.886
C09067=1152.860,135.105,-56.391,-178.784,6.740,148.885
C09068=1152.856,135.355,-56.410,-178.782,6.742,148.885
C09069=1152.851,135.604,-56.431,-178.779,6.743,148.885
C09070=1152.847,135.853,-56.451,-178.776,6.745,148.884
C09071=1152.842,136.102,-56.471,-178.773,6.747,148.884
C09072=1152.837,136.352,-56.492,-178.770,6.749,148.883
C09073=1152.832,136.601,-56.512,-178.767,6.751,148.883
C09074=1152.828,136.850,-56.532,-178.765,6.753,148.883
C09075=1152.823,137.099,-56.552,-178.762,6.755,148.882
C09076=1152.818,137.348,-56.573,-178.759,6.756,148.882
C09077=1152.813,137.597,-56.593,-178.757,6.758,148.881
C09078=1152.808,137.846,-56.613,-178.754,6.760,148.881
C09079=1152.803,138.095,-56.634,-178.751,6.761,148.881
C09080=1152.799,138.344,-56.654,-178.748,6.763,148.880
C09081=1152.794,138.593,-56.675,-178.746,6.765,148.880
C09082=1152.790,138.842,-56.695,-178.743,6.767,148.879
C09083=1152.784,139.092,-56.715,-178.740,6.768,148.879
C09084=1152.780,139.341,-56.736,-178.738,6.770,148.879
C09085=1152.775,139.590,-56.756,-178.735,6.772,148.878
C09086=1152.770,139.839,-56.777,-178.732,6.773,148.878
C09087=1152.766,140.088,-56.797,-178.729,6.776,148.878
C09088=1152.761,140.337,-56.818,-178.726,6.778,148.877
C09089=1152.756,140.587,-56.839,-178.723,6.779,148.877
C09090=1152.752,140.835,-56.859,-178.721,6.781,148.876
C09091=1152.747,141.085,-56.880,-178.718,6.783,148.876
C09092=1152.742,141.334,-56.900,-178.715,6.785,148.876
C09093=1152.737,141.583,-56.920,-178.713,6.786,148.875
C09094=1152.732,141.832,-56.941,-178.710,6.788,148.875
C09095=1152.728,142.081,-56.961,-178.707,6.790,148.874
C09096=1152.723,142.331,-56.982,-178.704,6.791,148.874
C09097=1152.718,142.580,-57.003,-178.702,6.794,148.874
C09098=1152.714,142.829,-57.023,-178.699,6.796,148.874
C09099=1152.709,143.078,-57.044,-178.696,6.798,148.873
C09100=1152.704,143.327,-57.064,-178.694,6.799,148.873
C09101=1152.699,143.576,-57.085,-178.691,6.801,148.872
C09102=1152.695,143.825,-57.106,-178.688,6.803,148.872
C09103=1152.690,144.074,-57.127,-178.685,6.805,148.872
C09104=1152.685,144.323,-57.148,-178.683,6.806,148.871
C09105=1152.680,144.572,-57.169,-178.680,6.808,148.871
C09106=1152.676,144.821,-57.189,-178.677,6.810,148.870
C09107=1152.671,145.071,-57.210,-178.674,6.812,148.870
C09108=1152.667,145.320,-57.231,-178.671,6.814,148.870
C09109=1152.661,145.569,-57.252,-178.669,6.816,148.869
C09110=1152.657,145.818,-57.272,-178.666,6.817,148.869
C09111=1152.652,146.067,-57.293,-178.663,6.819,148.869
C09112=1152.648,146.316,-57.314,-178.660,6.821,148.868
C09113=1152.642,146.565,-57.335,-178.658,6.823,148.868
C09114=1152.638,146.814,-57.356,-178.654,6.825,148.867
C09115=1152.633,147.063,-57.376,-178.652,6.827,148.867
C09116=1152.628,147.312,-57.397,-178.649,6.829,148.867
C09117=1152.624,147.561,-57.419,-178.646,6.830,148.866
C09118=1152.619,147.811,-57.440,-178.644,6.832,148.866
C09119=1152.615,148.059,-57.460,-178.641,6.834,148.866
C09120=1152.609,148.309,-57.481,-178.639,6.836,148.865
C09121=1152.605,148.557,-57.502,-178.636,6.838,148.865
C09122=1152.600,148.806,-57.523,-178.633,6.840,148.865
C09123=1152.595,149.056,-57.544,-178.630,6.842,148.864
C09124=1152.590,149.305,-57.565,-178.627,6.844,148.864
C09125=1152.586,149.554,-57.587,-178.625,6.845,148.863
C09126=1152.581,149.803,-57.608,-178.622,6.847,148.863
C09127=1152.577,150.052,-57.628,-178.619,6.849,148.863
C09128=1152.572,150.301,-57.650,-178.616,6.851,148.862
C09129=1152.567,150.550,-57.671,-178.613,6.853,148.862
C09130=1152.563,150.800,-57.691,-178.610,6.855,148.862
C09131=1152.558,151.048,-57.713,-178.608,6.856,148.861
C09132=1152.553,151.298,-57.734,-178.606,6.859,148.861
C09133=1152.548,151.546,-57.756,-178.603,6.860,148.861
C09134=1152.543,151.795,-57.776,-178.600,6.863,148.860
C09135=1152.538,152.044,-57.797,-178.597,6.865,148.860
C09136=1152.534,152.294,-57.819,-178.594,6.866,148.859
C09137=1152.529,152.543,-57.839,-178.591,6.868,148.859
C09138=1152.525,152.791,-57.861,-178.589,6.870,148.859
C09139=1152.519,153.041,-57.882,-178.586,6.871,148.858
C09140=1152.515,153.290,-57.904,-178.583,6.874,148.858
C09141=1152.511,153.539,-57.925,-178.580,6.876,148.858
C09142=1152.506,153.788,-57.946,-178.578,6.878,148.857
C09143=1152.501,154.037,-57.967,-178.575,6.880,148.857
C09144=1152.496,154.286,-57.989,-178.572,6.881,148.857
C09145=1152.491,154.535,-58.010,-178.569,6.884,148.856
C09146=1152.487,154.784,-58.031,-178.566,6.886,148.856
C09147=1152.482,155.033,-58.052,-178.564,6.887,148.856
C09148=1152.478,155.282,-58.074,-178.561,6.889,148.855
C09149=1152.473,155.531,-58.096,-178.558,6.891,148.855
C09150=1152.468,155.780,-58.117,-178.555,6.893,148.854
C09151=1152.463,156.029,-58.139,-178.553,6.895,148.854
C09152=1152.459,156.278,-58.159,-178.550,6.897,148.854
